REGION Network 21: PM1 Count & CycleTime / PM19 Count & CycleTime
   RUNG wire#powerrail
      #PM19CountCycleTime(iAlwaysOn := #iAlwaysOn, iProcessStart := "ST10_PM".Num[19].ProcessStart, iProcessComplete := "ST10_PM".Num[19].ProcessComplete, iProcessResult := "ST10_PM".Num[19].ProcessResult, ioCount := "ST10_PMCountCycleTime".PM[19].Count, ioTotalCycleTime := "ST10_PMCountCycleTime".PM[19].TotalCycleTime, ioMachineCycleTime := "ST10_PMCountCycleTime".PM[19].MachineCycleTime)
   END_RUNG
   // the same network as SCL:
   #PM19CountCycleTime(iAlwaysOn := #iAlwaysOn,   // "Count_CycleTime_V3"
                       iProcessStart := "ST10_PM".Num[19].ProcessStart,
                       iProcessComplete := "ST10_PM".Num[19].ProcessComplete,
                       iProcessResult := "ST10_PM".Num[19].ProcessResult,
                       ioCount := "ST10_PMCountCycleTime".PM[19].Count,
                       ioTotalCycleTime := "ST10_PMCountCycleTime".PM[19].TotalCycleTime,
                       ioMachineCycleTime := "ST10_PMCountCycleTime".PM[19].MachineCycleTime);
END_REGION

REGION Network 22: PM2 Count & CycleTime / PM20 Count & CycleTime
   RUNG wire#powerrail
      #PM20CountCycleTime(iAlwaysOn := #iAlwaysOn, iProcessStart := "ST10_PM".Num[20].ProcessStart, iProcessComplete := "ST10_PM".Num[20].ProcessComplete, iProcessResult := "ST10_PM".Num[20].ProcessResult, ioCount := "ST10_PMCountCycleTime".PM[20].Count, ioTotalCycleTime := "ST10_PMCountCycleTime".PM[20].TotalCycleTime, ioMachineCycleTime := "ST10_PMCountCycleTime".PM[20].MachineCycleTime)
   END_RUNG
   // the same network as SCL:
   #PM20CountCycleTime(iAlwaysOn := #iAlwaysOn,   // "Count_CycleTime_V3"
                       iProcessStart := "ST10_PM".Num[20].ProcessStart,
                       iProcessComplete := "ST10_PM".Num[20].ProcessComplete,
                       iProcessResult := "ST10_PM".Num[20].ProcessResult,
                       ioCount := "ST10_PMCountCycleTime".PM[20].Count,
                       ioTotalCycleTime := "ST10_PMCountCycleTime".PM[20].TotalCycleTime,
                       ioMachineCycleTime := "ST10_PMCountCycleTime".PM[20].MachineCycleTime);
END_REGION

REGION Network 23: PM2 Count & CycleTime / PM21 Count & CycleTime
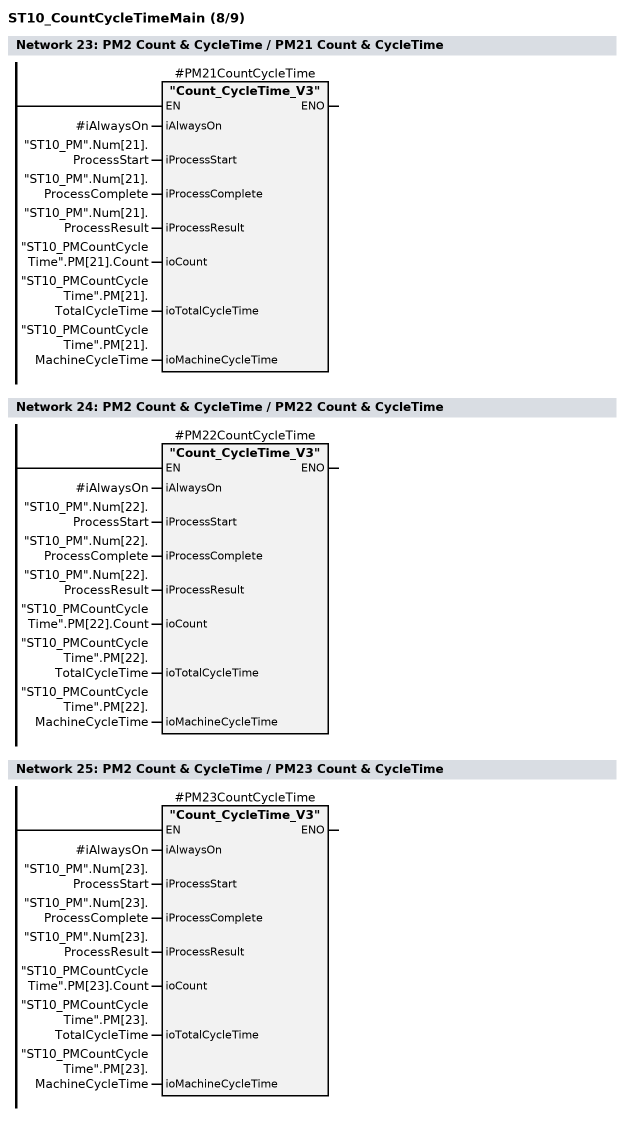
   RUNG wire#powerrail
      #PM21CountCycleTime(iAlwaysOn := #iAlwaysOn, iProcessStart := "ST10_PM".Num[21].ProcessStart, iProcessComplete := "ST10_PM".Num[21].ProcessComplete, iProcessResult := "ST10_PM".Num[21].ProcessResult, ioCount := "ST10_PMCountCycleTime".PM[21].Count, ioTotalCycleTime := "ST10_PMCountCycleTime".PM[21].TotalCycleTime, ioMachineCycleTime := "ST10_PMCountCycleTime".PM[21].MachineCycleTime)
   END_RUNG
   // the same network as SCL:
   #PM21CountCycleTime(iAlwaysOn := #iAlwaysOn,   // "Count_CycleTime_V3"
                       iProcessStart := "ST10_PM".Num[21].ProcessStart,
                       iProcessComplete := "ST10_PM".Num[21].ProcessComplete,
                       iProcessResult := "ST10_PM".Num[21].ProcessResult,
                       ioCount := "ST10_PMCountCycleTime".PM[21].Count,
                       ioTotalCycleTime := "ST10_PMCountCycleTime".PM[21].TotalCycleTime,
                       ioMachineCycleTime := "ST10_PMCountCycleTime".PM[21].MachineCycleTime);
END_REGION

REGION Network 24: PM2 Count & CycleTime / PM22 Count & CycleTime
   RUNG wire#powerrail
      #PM22CountCycleTime(iAlwaysOn := #iAlwaysOn, iProcessStart := "ST10_PM".Num[22].ProcessStart, iProcessComplete := "ST10_PM".Num[22].ProcessComplete, iProcessResult := "ST10_PM".Num[22].ProcessResult, ioCount := "ST10_PMCountCycleTime".PM[22].Count, ioTotalCycleTime := "ST10_PMCountCycleTime".PM[22].TotalCycleTime, ioMachineCycleTime := "ST10_PMCountCycleTime".PM[22].MachineCycleTime)
   END_RUNG
   // the same network as SCL:
   #PM22CountCycleTime(iAlwaysOn := #iAlwaysOn,   // "Count_CycleTime_V3"
                       iProcessStart := "ST10_PM".Num[22].ProcessStart,
                       iProcessComplete := "ST10_PM".Num[22].ProcessComplete,
                       iProcessResult := "ST10_PM".Num[22].ProcessResult,
                       ioCount := "ST10_PMCountCycleTime".PM[22].Count,
                       ioTotalCycleTime := "ST10_PMCountCycleTime".PM[22].TotalCycleTime,
                       ioMachineCycleTime := "ST10_PMCountCycleTime".PM[22].MachineCycleTime);
END_REGION

REGION Network 25: PM2 Count & CycleTime / PM23 Count & CycleTime
   RUNG wire#powerrail
      #PM23CountCycleTime(iAlwaysOn := #iAlwaysOn, iProcessStart := "ST10_PM".Num[23].ProcessStart, iProcessComplete := "ST10_PM".Num[23].ProcessComplete, iProcessResult := "ST10_PM".Num[23].ProcessResult, ioCount := "ST10_PMCountCycleTime".PM[23].Count, ioTotalCycleTime := "ST10_PMCountCycleTime".PM[23].TotalCycleTime, ioMachineCycleTime := "ST10_PMCountCycleTime".PM[23].MachineCycleTime)
   END_RUNG
   // the same network as SCL:
   #PM23CountCycleTime(iAlwaysOn := #iAlwaysOn,   // "Count_CycleTime_V3"
                       iProcessStart := "ST10_PM".Num[23].ProcessStart,
                       iProcessComplete := "ST10_PM".Num[23].ProcessComplete,
                       iProcessResult := "ST10_PM".Num[23].ProcessResult,
                       ioCount := "ST10_PMCountCycleTime".PM[23].Count,
                       ioTotalCycleTime := "ST10_PMCountCycleTime".PM[23].TotalCycleTime,
                       ioMachineCycleTime := "ST10_PMCountCycleTime".PM[23].MachineCycleTime);
END_REGION

REGION Network 26: PM2 Count & CycleTime / PM24 Count & CycleTime
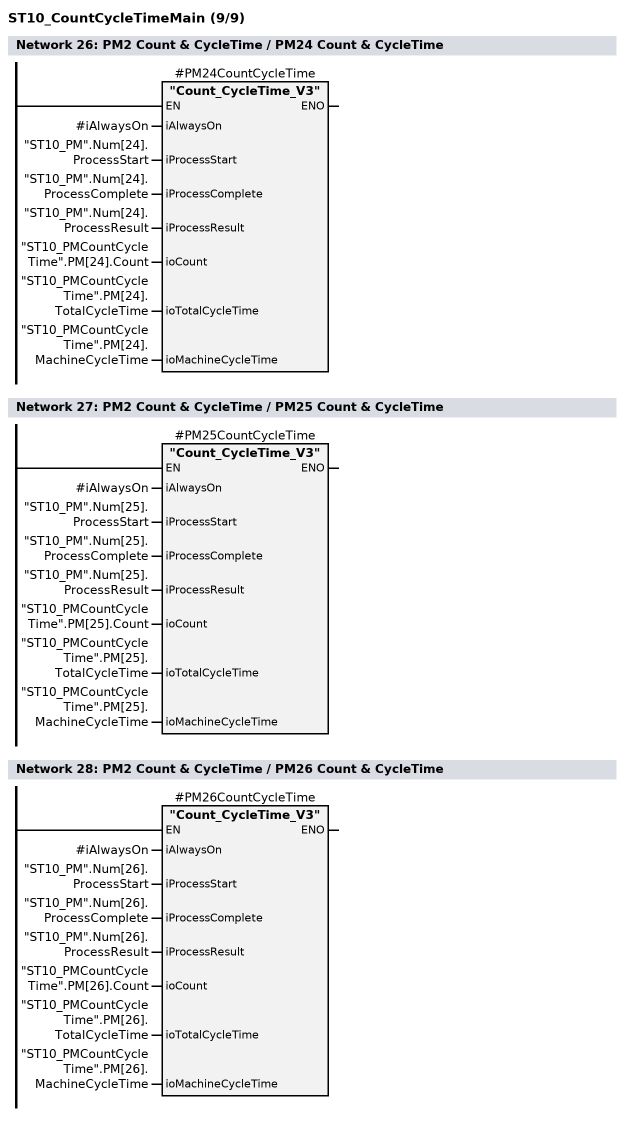
   RUNG wire#powerrail
      #PM24CountCycleTime(iAlwaysOn := #iAlwaysOn, iProcessStart := "ST10_PM".Num[24].ProcessStart, iProcessComplete := "ST10_PM".Num[24].ProcessComplete, iProcessResult := "ST10_PM".Num[24].ProcessResult, ioCount := "ST10_PMCountCycleTime".PM[24].Count, ioTotalCycleTime := "ST10_PMCountCycleTime".PM[24].TotalCycleTime, ioMachineCycleTime := "ST10_PMCountCycleTime".PM[24].MachineCycleTime)
   END_RUNG
   // the same network as SCL:
   #PM24CountCycleTime(iAlwaysOn := #iAlwaysOn,   // "Count_CycleTime_V3"
                       iProcessStart := "ST10_PM".Num[24].ProcessStart,
                       iProcessComplete := "ST10_PM".Num[24].ProcessComplete,
                       iProcessResult := "ST10_PM".Num[24].ProcessResult,
                       ioCount := "ST10_PMCountCycleTime".PM[24].Count,
                       ioTotalCycleTime := "ST10_PMCountCycleTime".PM[24].TotalCycleTime,
                       ioMachineCycleTime := "ST10_PMCountCycleTime".PM[24].MachineCycleTime);
END_REGION

REGION Network 27: PM2 Count & CycleTime / PM25 Count & CycleTime
   RUNG wire#powerrail
      #PM25CountCycleTime(iAlwaysOn := #iAlwaysOn, iProcessStart := "ST10_PM".Num[25].ProcessStart, iProcessComplete := "ST10_PM".Num[25].ProcessComplete, iProcessResult := "ST10_PM".Num[25].ProcessResult, ioCount := "ST10_PMCountCycleTime".PM[25].Count, ioTotalCycleTime := "ST10_PMCountCycleTime".PM[25].TotalCycleTime, ioMachineCycleTime := "ST10_PMCountCycleTime".PM[25].MachineCycleTime)
   END_RUNG
   // the same network as SCL:
   #PM25CountCycleTime(iAlwaysOn := #iAlwaysOn,   // "Count_CycleTime_V3"
                       iProcessStart := "ST10_PM".Num[25].ProcessStart,
                       iProcessComplete := "ST10_PM".Num[25].ProcessComplete,
                       iProcessResult := "ST10_PM".Num[25].ProcessResult,
                       ioCount := "ST10_PMCountCycleTime".PM[25].Count,
                       ioTotalCycleTime := "ST10_PMCountCycleTime".PM[25].TotalCycleTime,
                       ioMachineCycleTime := "ST10_PMCountCycleTime".PM[25].MachineCycleTime);
END_REGION

REGION Network 28: PM2 Count & CycleTime / PM26 Count & CycleTime
   RUNG wire#powerrail
      #PM26CountCycleTime(iAlwaysOn := #iAlwaysOn, iProcessStart := "ST10_PM".Num[26].ProcessStart, iProcessComplete := "ST10_PM".Num[26].ProcessComplete, iProcessResult := "ST10_PM".Num[26].ProcessResult, ioCount := "ST10_PMCountCycleTime".PM[26].Count, ioTotalCycleTime := "ST10_PMCountCycleTime".PM[26].TotalCycleTime, ioMachineCycleTime := "ST10_PMCountCycleTime".PM[26].MachineCycleTime)
   END_RUNG
   // the same network as SCL:
   #PM26CountCycleTime(iAlwaysOn := #iAlwaysOn,   // "Count_CycleTime_V3"
                       iProcessStart := "ST10_PM".Num[26].ProcessStart,
                       iProcessComplete := "ST10_PM".Num[26].ProcessComplete,
                       iProcessResult := "ST10_PM".Num[26].ProcessResult,
                       ioCount := "ST10_PMCountCycleTime".PM[26].Count,
                       ioTotalCycleTime := "ST10_PMCountCycleTime".PM[26].TotalCycleTime,
                       ioMachineCycleTime := "ST10_PMCountCycleTime".PM[26].MachineCycleTime);
END_REGION
END_FUNCTION_BLOCK

FUNCTION_BLOCK "Count_CycleTime"   // FB3002, SCL
TITLE = Count_CycleTime
{ S7_Optimized_Access := 'TRUE' }
AUTHOR : STD
FAMILY : RCS
VERSION : 18.0
// 1.count
// 2.cycle time
// stored: AutoNumber false, MemoryReserve 100, SetENOAutomatically false, UDAEnableTagReadback true
   VAR_INPUT
      iAlwaysOn : Bool;
      iRun : Bool;
      iManualMode : Bool;
      iAutoMode : Bool;
      iAutoRunning : Bool;
      iProcessStart : Bool;
      iProcessComplete : Bool;
      iProcessResult : DInt;
   END_VAR
   VAR_IN_OUT
      ioCount : "RCS_SysCount_V1";
      ioTotalCycleTime : "RCS_SysCycleTime_V1";
      ioMachineCycleTime : "RCS_SysCycleTime_V1";
   END_VAR
   VAR
      sFlow : Struct
         pls : Array[0..15] of Bool;
         sDTStart : Date_And_Time;
         sDTRes : Date_And_Time;
         sDTOld : Date_And_Time;
         sDTRuntime : Date_And_Time;
         sDTRunning : Date_And_Time;
         sDTCurrent : Date_And_Time;
         Run_Minute : Int;
         Run_Hour : Int;
         Run_Day : Int;
         AutoRun_Minute : Int;
         AutoRun_Hour : Int;
         AutoRun_Day : Int;
      END_STRUCT;
   END_VAR
   VAR_TEMP
      tStart : Bool;
      tStop : Bool;
      tAutorunning : Bool;
      tpt : Int;
      tpRet : Int;
      tpResult : Time;
      tDint : DInt;
      tReal : Array[0..1] of Real;
   END_VAR
BEGIN
   (*############################################################
      RUHLAMAT SUZHOU ELEC.STD.
      Copyright (c) 2017. All rights reserved.    

      NAME OF FUNCTION BLOCK:         Count_CycleTimeV2.0
      VERSION NUMBER:                 V2.0
      COMPOSER:                       Ming.Jiang

      LAST CHANGE:                    13.April.2017
      Comment by Ming.Jiang 

      #RET_VALUE:


      #Alert Value:



      -----------------------------------------------------
      Date        Name      Version           Activity                                                                              

   ############################################################*)

   #tStart := #iProcessStart AND NOT #sFlow.pls[0];
   #sFlow.pls[0] := #iProcessStart;
   #tStop := #iProcessComplete AND NOT #sFlow.pls[1];
   #sFlow.pls[1] := #iProcessComplete;
   #tAutorunning := #iAutoMode AND #iAutoRunning AND NOT #sFlow.pls[2];
   #sFlow.pls[2] := #iAutoRunning AND #iAutoMode;

   IF #tAutorunning THEN
       #tpRet := RD_SYS_T(#sFlow.sDTOld);
   END_IF;

   //Machine Cycle time
   IF #iAutoMode AND NOT #iManualMode AND #iAutoRunning THEN
       IF #tStart THEN
           #tpRet := RD_SYS_T(#sFlow.sDTStart);
       END_IF;
       IF #tStop THEN

           //MachineTime
           #ioMachineCycleTime.No[21] := 0.0;
           #tpRet := RD_SYS_T(#sFlow.sDTRes);
           #tReal[0] := DINT_TO_REAL(TIME_TO_DINT(T_DIFF(IN1 := #sFlow.sDTRes, IN2 :=#sFlow.sDTStart )));
           #ioMachineCycleTime.No[0] :=  #tReal[0]/1000.0;

           //TotalTime
           #ioTotalCycleTime.No[21] := 0.0;
           #tReal[1] := DINT_TO_REAL(TIME_TO_DINT(T_DIFF(IN1 := #sFlow.sDTRes, IN2 := #sFlow.sDTOld)));
           #tpRet := RD_SYS_T(#sFlow.sDTOld);
           #ioTotalCycleTime.No[0] := #tReal[1]/1000.0;
           FOR #tpt := 20 TO 1 BY -1  DO
               //MachineTime
               #ioMachineCycleTime.No[#tpt] := #ioMachineCycleTime.No[#tpt - 1];
               #ioMachineCycleTime.No[21] := #ioMachineCycleTime.No[21] + #ioMachineCycleTime.No[#tpt];
               //totalCycleTime
               #ioTotalCycleTime.No[#tpt] := #ioTotalCycleTime.No[#tpt - 1];
               #ioTotalCycleTime.No[21] := #ioTotalCycleTime.No[21] + #ioTotalCycleTime.No[#tpt];
           END_FOR;
           //MachineTime
           #ioMachineCycleTime.No[21] := #ioMachineCycleTime.No[21] / 20.0;
           //totalCycleTime
           #ioTotalCycleTime.No[21] := #ioTotalCycleTime.No[21] / 20.0;

           //Count-------------------------------------------------------//
           IF #iProcessResult = 400 THEN
               #ioCount.OK[0] := #ioCount.OK[0] + 1;
               #ioCount.OKHolding := #ioCount.OKHolding + 1;
           END_IF;
           IF #iProcessResult > 400  THEN
               #ioCount.NG[0] := #ioCount.NG[0] + 1;
               #ioCount.NGHolding:=#ioCount.NGHolding+1;
           END_IF;
           IF #iProcessResult >=400  THEN
               #ioCount.Total := #ioCount.Total + 1;
           END_IF;
           #ioCount.OKHolding := #ioCount.OKHolding + 1;

           CASE #iProcessResult OF
               401:  //NG1
                   #ioCount.NG[1] := #ioCount.NG[1] + 1;
               402:  //NG1uuuuuuuuuuuuuuuuuuuuuuuuuuuuuuuuuuuuuuuuuuuuuuuu
                   #ioCount.NG[2] := #ioCount.NG[2] + 1;
               403:  //NG1uuuuu
                   #ioCount.NG[3] := #ioCount.NG[3] + 1;
               404:  //NG1
                   #ioCount.NG[4] := #ioCount.NG[4] + 1;
               405:  //NG1
                   #ioCount.NG[5] := #ioCount.NG[5] + 1;
               406:  //NG1
                   #ioCount.NG[6] := #ioCount.NG[6] + 1;
               407:  //NG1
                   #ioCount.NG[7] := #ioCount.NG[7] + 1;
               408:  //NG1
                   #ioCount.NG[8] := #ioCount.NG[8] + 1;
               409:  //NG1
                   #ioCount.NG[9] := #ioCount.NG[9] + 1;

           END_CASE;
       END_IF;

   END_IF;
   //clear 
   IF #ioCount.ClearOK AND NOT #sFlow.pls[3] THEN
       #ioCount.OK[0] := 0;

   END_IF;
   #sFlow.pls[3] := #ioCount.ClearOK;
   IF #ioCount.ClearNG AND NOT #sFlow.pls[4] THEN
       FOR #tpt := 0 TO 9 DO
            #ioCount.NG[#tpt] := 0;
        END_FOR;
   END_IF;
   #sFlow.pls[4] := #ioCount.ClearNG;
   IF #ioCount.ClearTotal AND NOT #sFlow.pls[5] THEN
       #ioCount.Total := 0;

   END_IF;
   #sFlow.pls[5] := #ioCount.ClearTotal;
   //Runtime

   IF #iAutoRunning AND NOT #sFlow.pls[6] THEN
       #tpRet := RD_SYS_T(#sFlow.sDTRunning);

   END_IF;
   #sFlow.pls[6] := #iAutoRunning;
   #tpRet := RD_SYS_T(#sFlow.sDTCurrent);
   IF #iAutoRunning THEN
       #tDint := TIME_TO_DINT(T_DIFF(IN1 := #sFlow.sDTCurrent, IN2 := #sFlow.sDTRunning));
       #tReal[0] := DINT_TO_REAL(#tDint) / 1000.0;
       #sFlow.AutoRun_Day := REAL_TO_INT(#tReal[0] / 86400.0);
       #sFlow.AutoRun_Hour := (REAL_TO_DINT(#tReal[0]) MOD 86400) / 3600;
       #sFlow.AutoRun_Minute := ((REAL_TO_DINT(#tReal[0]) MOD 86400) MOD 3600) / 60;
   END_IF;

   //Runtime
   IF #iRun AND NOT #sFlow.pls[7] THEN
       #tpRet := RD_SYS_T(#sFlow.sDTRuntime);
   END_IF;
   #sFlow.pls[7] := #iRun;
   IF #iRun THEN
       #tDint := TIME_TO_DINT(T_DIFF(IN1 := #sFlow.sDTCurrent, IN2 :=#sFlow.sDTRuntime ));
       #tReal[0] := DINT_TO_REAL(#tDint) / 1000.0;
       #sFlow.Run_Day := REAL_TO_INT(#tReal[0] / 86400.0);
       #sFlow.Run_Hour := (REAL_TO_DINT(#tReal[0]) MOD 86400) / 3600;
       #sFlow.Run_Minute := ((REAL_TO_DINT(#tReal[0]) MOD 86400) MOD 3600) / 60;
   END_IF;
END_FUNCTION_BLOCK

FUNCTION_BLOCK "Count_CycleTime_V3"   // FB3003, SCL
TITLE = Count_CycleTime
{ S7_Optimized_Access := 'TRUE' }
AUTHOR : STD
FAMILY : RCS
VERSION : 18.0
// 1.count
// 2.cycle time
// stored: AutoNumber false, MemoryReserve 100, SetENOAutomatically false, UDAEnableTagReadback true
   VAR_INPUT
      iAlwaysOn : Bool;
      iProcessStart : Bool;
      iProcessComplete : Bool;
      iProcessResult : DInt;
   END_VAR
   VAR_IN_OUT
      ioCount : "RCS_SysCount_V1";
      ioTotalCycleTime : "RCS_SysCycleTime_V1";
      ioMachineCycleTime : "RCS_SysCycleTime_V1";
   END_VAR
   VAR
      sFlow : Struct
         pls : Array[0..15] of Bool;
         sDTStart : Date_And_Time;
         sDTRes : Date_And_Time;
         sDTOld : Date_And_Time;
         sDTRuntime : Date_And_Time;
         sDTRunning : Date_And_Time;
         sDTCurrent : Date_And_Time;
         Run_Minute : Int;
         Run_Hour : Int;
         Run_Day : Int;
         AutoRun_Minute : Int;
         AutoRun_Hour : Int;
         AutoRun_Day : Int;
      END_STRUCT;
   END_VAR
   VAR_TEMP
      tStart : Bool;
      tStop : Bool;
      tAutorunning : Bool;
      tpt : Int;
      tpRet : Int;
      tpResult : Time;
      tDint : DInt;
      tReal : Array[0..1] of Real;
   END_VAR
BEGIN
   (*############################################################
      RUHLAMAT SUZHOU ELEC.STD.
      Copyright (c) 2017. All rights reserved.    

      NAME OF FUNCTION BLOCK:         Count_CycleTimeV2.0
      VERSION NUMBER:                 V2.0
      COMPOSER:                       Ming.Jiang

      LAST CHANGE:                    13.April.2017
      Comment by Ming.Jiang 

      #RET_VALUE:


      #Alert Value:



      -----------------------------------------------------
      Date        Name      Version           Activity                                                                              

   ############################################################*)

   #tStart := #iProcessStart AND NOT #sFlow.pls[0];
   #sFlow.pls[0] := #iProcessStart;
   #tStop := #iProcessComplete AND NOT #sFlow.pls[1];
   #sFlow.pls[1] := #iProcessComplete;

   // IF #tStop THEN
   //     #tpRet := RD_SYS_T(#sFlow.sDTOld);
   // END_IF;

   //Machine Cycle time
   IF TRUE THEN
       IF #tStart THEN
           #tpRet := RD_SYS_T(#sFlow.sDTStart);
       END_IF;
       IF #tStop THEN

           //MachineTime
           #ioMachineCycleTime.No[21] := 0.0;
           #tpRet := RD_SYS_T(#sFlow.sDTRes);
           #tReal[0] := DINT_TO_REAL(TIME_TO_DINT(T_DIFF(IN1 := #sFlow.sDTRes, IN2 :=#sFlow.sDTStart )));
           #ioMachineCycleTime.No[0] :=  #tReal[0]/1000.0;

           //TotalTime
           #ioTotalCycleTime.No[21] := 0.0;
           #tReal[1] := DINT_TO_REAL(TIME_TO_DINT(T_DIFF(IN1 := #sFlow.sDTRes, IN2 := #sFlow.sDTOld)));
           #tpRet := RD_SYS_T(#sFlow.sDTOld);
           #ioTotalCycleTime.No[0] := #tReal[1]/1000.0;
           FOR #tpt := 20 TO 1 BY -1  DO
               //MachineTime
               #ioMachineCycleTime.No[#tpt] := #ioMachineCycleTime.No[#tpt - 1];
               #ioMachineCycleTime.No[21] := #ioMachineCycleTime.No[21] + #ioMachineCycleTime.No[#tpt];
               //totalCycleTime
               #ioTotalCycleTime.No[#tpt] := #ioTotalCycleTime.No[#tpt - 1];
               #ioTotalCycleTime.No[21] := #ioTotalCycleTime.No[21] + #ioTotalCycleTime.No[#tpt];
           END_FOR;
           //MachineTime
           #ioMachineCycleTime.No[21] := #ioMachineCycleTime.No[21] / 20.0;
           //totalCycleTime
           #ioTotalCycleTime.No[21] := #ioTotalCycleTime.No[21] / 20.0;

           //Count-------------------------------------------------------//
           IF #iProcessResult = 400 THEN
               #ioCount.OK[0] := #ioCount.OK[0] + 1;
               #ioCount.OKHolding := #ioCount.OKHolding + 1;
           END_IF;
           IF #iProcessResult >400 THEN
               #ioCount.NG[0] := #ioCount.NG[0] + 1;
               #ioCount.NGHolding:=#ioCount.NGHolding+1;
           END_IF;
           IF #iProcessResult >=400 THEN
               #ioCount.Total := #ioCount.Total + 1;
           END_IF;
           #ioCount.OKHolding := #ioCount.OKHolding + 1;

           CASE #iProcessResult OF
               401:  //NG1
                   #ioCount.NG[1] := #ioCount.NG[1] + 1;
               402:  //NG1uuuuuuuuuuuuuuuuuuuuuuuuuuuuuuuuuuuuuuuuuuuuuuuu
                   #ioCount.NG[2] := #ioCount.NG[2] + 1;
               403:  //NG1uuuuu
                   #ioCount.NG[3] := #ioCount.NG[3] + 1;
               404:  //NG1
                   #ioCount.NG[4] := #ioCount.NG[4] + 1;
               405:  //NG1
                   #ioCount.NG[5] := #ioCount.NG[5] + 1;
               406:  //NG1
                   #ioCount.NG[6] := #ioCount.NG[6] + 1;
               407:  //NG1
                   #ioCount.NG[7] := #ioCount.NG[7] + 1;
               408:  //NG1
                   #ioCount.NG[8] := #ioCount.NG[8] + 1;
               409:  //NG1
                   #ioCount.NG[9] := #ioCount.NG[9] + 1;

           END_CASE;
       END_IF;

   END_IF;
   //clear 
   IF #ioCount.ClearOK AND NOT #sFlow.pls[3] THEN
       #ioCount.OK[0] := 0;

   END_IF;
   #sFlow.pls[3] := #ioCount.ClearOK;
   IF #ioCount.ClearNG AND NOT #sFlow.pls[4] THEN
       FOR #tpt := 0 TO 9 DO
            #ioCount.NG[#tpt] := 0;
        END_FOR;
   END_IF;
   #sFlow.pls[4] := #ioCount.ClearNG;
   IF #ioCount.ClearTotal AND NOT #sFlow.pls[5] THEN
       #ioCount.Total := 0;

   END_IF;
   #sFlow.pls[5] := #ioCount.ClearTotal;
END_FUNCTION_BLOCK

FUNCTION_BLOCK "SystemMode"   // FB3000, LAD
TITLE = SystemMode_FB
{ S7_Optimized_Access := 'TRUE' }
AUTHOR : STD
FAMILY : RCS
VERSION : 2.0
// stored: AutoNumber false, MemoryReserve 100, SetENOAutomatically false
   VAR_INPUT
      iPLCRestarted : Bool;
      iEstopAllOK { ExternalAccessible := 'False'; ExternalVisible := 'False'; ExternalWritable := 'False'} : Bool;   // 急停按钮
      iResetFault { ExternalAccessible := 'False'; ExternalVisible := 'False'; ExternalWritable := 'False'} : Bool;   // 故障复位按钮
      iModeSelectType { ExternalAccessible := 'False'; ExternalVisible := 'False'; ExternalWritable := 'False'} : Bool;   // 0=key switch / 1= HMI button
      iManual { ExternalAccessible := 'False'; ExternalVisible := 'False'; ExternalWritable := 'False'} : Bool;   // Key switch signal,1=Manual / Key switch signal,1=Manual Mode
      iAuto { ExternalAccessible := 'False'; ExternalVisible := 'False'; ExternalWritable := 'False'} : Bool;   // Key switch signal,1=Auto / Key switch signal,1=Auto Mode
      iStep { ExternalAccessible := 'False'; ExternalVisible := 'False'; ExternalWritable := 'False'} : Bool;   // Step mode / Auto Step Mode
      iOneCycle : Bool;   // OneCycle / Auto One Cycle Mode
      iHMIModeSelect { ExternalAccessible := 'False'; ExternalVisible := 'False'; ExternalWritable := 'False'} : Int;   // HMI button signal,1=Manual / 2=Auto/3=OneCycle/4=Step / HMI button signal,1=Manual / 2=Auto / 3=Step / 4=OneCyc
      iControlOnMonitor { ExternalAccessible := 'False'; ExternalVisible := 'False'; ExternalWritable := 'False'} : Bool;   // 安全继电器ControlOn监控
      iSafetyDoor { ExternalAccessible := 'False'; ExternalVisible := 'False'; ExternalWritable := 'False'} : Bool;
      iLightCurtain { ExternalAccessible := 'False'; ExternalVisible := 'False'; ExternalWritable := 'False'} : Bool;
      iSafetyByPass : Bool;
      iMainPressureSwitch { ExternalAccessible := 'False'; ExternalVisible := 'False'; ExternalWritable := 'False'} : Bool;   // 主气源开关监控
      iFixtureOK { ExternalAccessible := 'False'; ExternalVisible := 'False'; ExternalWritable := 'False'} : Bool;   // fixture ok
      iChangeOverOK { ExternalAccessible := 'False'; ExternalVisible := 'False'; ExternalWritable := 'False'} : Bool;   // changer over is ok
      iInitializationOK { ExternalAccessible := 'False'; ExternalVisible := 'False'; ExternalWritable := 'False'} : Bool;   // initialization is ok
      iAllDeviceOK { ExternalAccessible := 'False'; ExternalVisible := 'False'; ExternalWritable := 'False'} : Bool;   // all device is ready
      iAlarmOn : Bool;   // 设备故障
      iFlowRun : Bool;   // 设备运行
   END_VAR
   VAR_OUTPUT
      oReset { ExternalAccessible := 'False'; ExternalVisible := 'False'; ExternalWritable := 'False'} : Bool;   // 系统复位信号
      oEStopOK { ExternalAccessible := 'False'; ExternalVisible := 'False'; ExternalWritable := 'False'} : Bool;   // 系统急停控制信号
      oManualMode { ExternalAccessible := 'False'; ExternalVisible := 'False'; ExternalWritable := 'False'} : Bool;   // 手动模式信号
      oAutoMode { ExternalAccessible := 'False'; ExternalVisible := 'False'; ExternalWritable := 'False'} : Bool;   // 自动模式信号
      oOneCycleMode : Bool;   // 单次循环
      oStepMode { ExternalAccessible := 'False'; ExternalVisible := 'False'; ExternalWritable := 'False'} : Bool;
      oRun { ExternalAccessible := 'False'; ExternalVisible := 'False'; ExternalWritable := 'False'} : Bool;   // 系统运行就绪信号 / Control On and all Safety function OK
      "oEnable alarm" : Bool;
      oControlON { ExternalAccessible := 'False'; ExternalVisible := 'False'; ExternalWritable := 'False'} : Bool;   // PowerON
      oMainPressureOK { ExternalAccessible := 'False'; ExternalVisible := 'False'; ExternalWritable := 'False'} : Bool;   // air pressure
      oSafetyDoorOK { ExternalAccessible := 'False'; ExternalVisible := 'False'; ExternalWritable := 'False'} : Bool;   // 安全门关闭
      oLightCurtainOK { ExternalAccessible := 'False'; ExternalVisible := 'False'; ExternalWritable := 'False'} : Bool;   // 光栅
      oReady : Bool;   // 用于流程控制 / In AutoMode and all condition ok, machine can auto running
      oMode { ExternalAccessible := 'False'; ExternalVisible := 'False'; ExternalWritable := 'False'} : Int;   // 0NA,1Manual, 2Auto, 3Step, 4OneCycle, 5Runn, 6Error
      oStatus : Int;   // 0NotReady, 1Ready, 2AutoRunning, 3EStop, 4Alarm
   END_VAR
   VAR
      sRunT { S7_SetPoint := 'True'} : TON_TIME;
      sPressureTOF { S7_SetPoint := 'True'} : TOF_TIME;
      sChangeOverTOF { S7_SetPoint := 'True'} : TOF_TIME;
      sChangeOverOK { S7_SetPoint := 'True'} : Bool;
   END_VAR
   VAR_TEMP
      tAlwaysOn : Bool;
   END_VAR
   VAR_TEMP   // added for the SCL form of the ladder/FBD networks
      _w1 : Bool;
      _w2 : Bool;
      _w3 : Bool;
   END_VAR
BEGIN

REGION Network 1: AlwaysOn
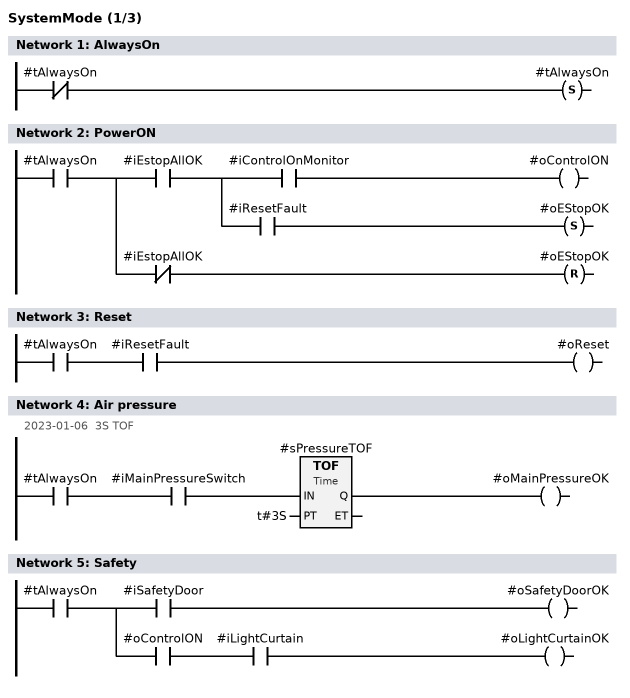
   RUNG wire#powerrail
      I_Contact( #tAlwaysOn )
      S_Coil( #tAlwaysOn )
   END_RUNG
   // the same network as SCL:
   IF NOT #tAlwaysOn THEN #tAlwaysOn := TRUE; END_IF;
END_REGION

REGION Network 2: PowerON
   RUNG wire#powerrail
      Contact( #tAlwaysOn )
      wire#w1
      Contact( #iEstopAllOK )
      wire#w2
      Contact( #iControlOnMonitor )
      Coil( #oControlON )
   END_RUNG
   RUNG wire#w2
      Contact( #iResetFault )
      S_Coil( #oEStopOK )
   END_RUNG
   RUNG wire#w1
      I_Contact( #iEstopAllOK )
      R_Coil( #oEStopOK )
   END_RUNG
   // the same network as SCL:
   #_w1 := #tAlwaysOn AND #iEstopAllOK;
   #oControlON := #_w1 AND #iControlOnMonitor;
   IF #_w1 AND #iResetFault THEN #oEStopOK := TRUE; END_IF;
   IF #tAlwaysOn AND NOT #iEstopAllOK THEN #oEStopOK := FALSE; END_IF;
END_REGION

REGION Network 3: Reset
   RUNG wire#powerrail
      Contact( #tAlwaysOn )
      Contact( #iResetFault )
      Coil( #oReset )
   END_RUNG
   // the same network as SCL:
   #oReset := #tAlwaysOn AND #iResetFault;
END_REGION

REGION Network 4: Air pressure
   // 2023-01-06  3S TOF
   RUNG wire#powerrail
      Contact( #tAlwaysOn )
      Contact( #iMainPressureSwitch )
      { S7_Templates := "time_type := Time" } #sPressureTOF.TOF(pt := t#3S, et =>)
      Coil( #oMainPressureOK )
   END_RUNG
   // the same network as SCL:
   #sPressureTOF(IN := #tAlwaysOn AND #iMainPressureSwitch, PT := t#3S);   // TOF
   #oMainPressureOK := #sPressureTOF.Q;
END_REGION

REGION Network 5: Safety
   RUNG wire#powerrail
      Contact( #tAlwaysOn )
      wire#w1
      Contact( #iSafetyDoor )
      Coil( #oSafetyDoorOK )
   END_RUNG
   RUNG wire#w1
      Contact( #oControlON )
      Contact( #iLightCurtain )
      Coil( #oLightCurtainOK )
   END_RUNG
   // the same network as SCL:
   #oSafetyDoorOK := #tAlwaysOn AND #iSafetyDoor;
   #oLightCurtainOK := #tAlwaysOn AND #oControlON AND #iLightCurtain;
END_REGION

REGION Network 6: Mode
   // 0NA,1Manual, 2Auto, 3Step, 4OneCycle, 5Runn, 6Error
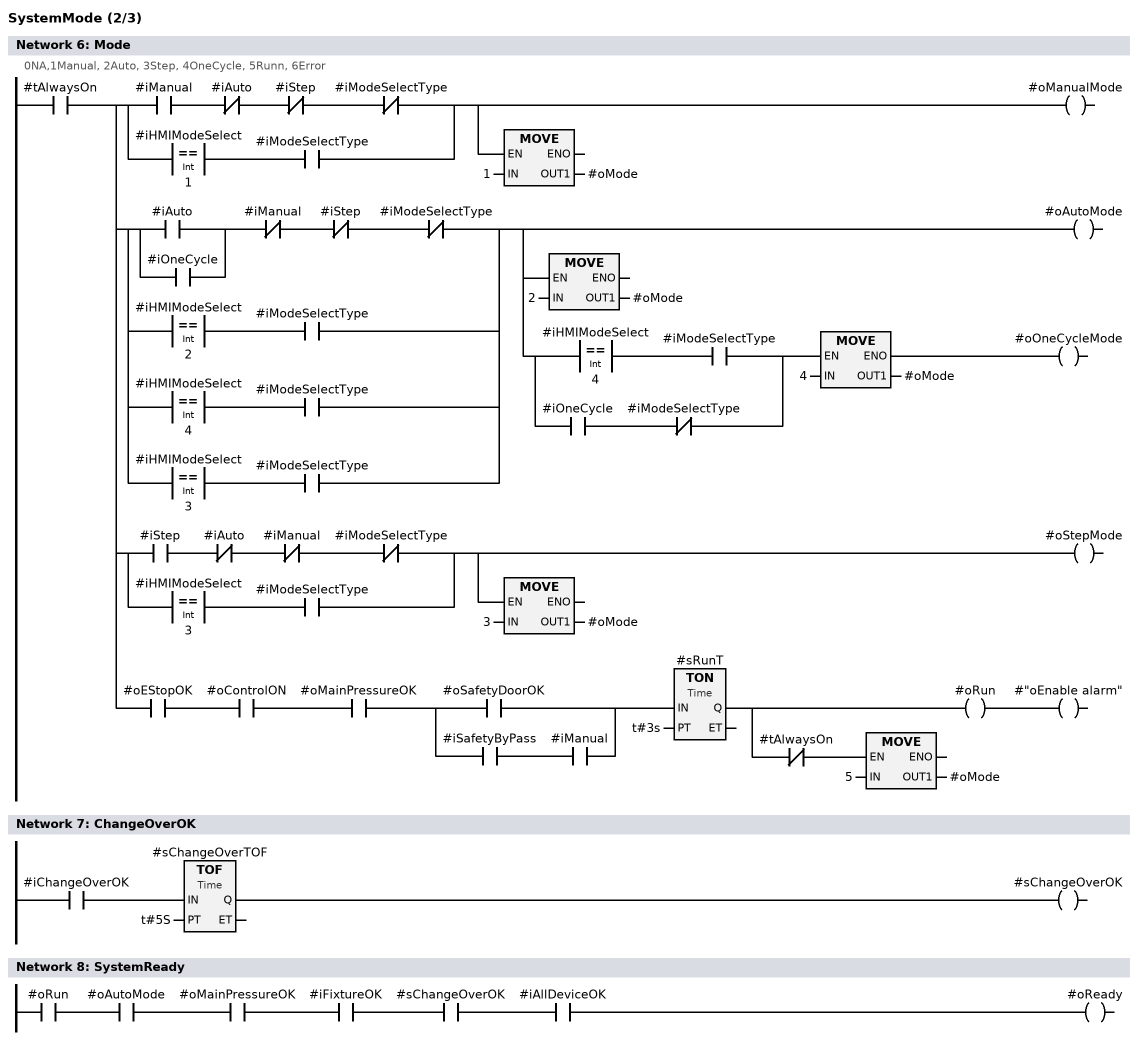
   RUNG wire#powerrail
      Contact( #tAlwaysOn )
      wire#w1
      Contact( #iManual )
      I_Contact( #iAuto )
      I_Contact( #iStep )
      I_Contact( #iModeSelectType )
      wire#w2
      Coil( #oManualMode )
   END_RUNG
   RUNG wire#w1
      { S7_Templates := "SrcType := Int" } EQ_Contact(in1 := #iHMIModeSelect, in2 := 1)
      Contact( #iModeSelectType )
   END_RUNG wire#w2
   RUNG wire#w2
      { S7_GenerateENO := "TRUE" } Move(in := 1, out1 => #oMode)
   END_RUNG
   RUNG wire#w1
      Contact( #iAuto )
      wire#w3
      I_Contact( #iManual )
      I_Contact( #iStep )
      I_Contact( #iModeSelectType )
      wire#w4
      Coil( #oAutoMode )
   END_RUNG
   RUNG wire#w1
      Contact( #iOneCycle )
   END_RUNG wire#w3
   RUNG wire#w1
      { S7_Templates := "SrcType := Int" } EQ_Contact(in1 := #iHMIModeSelect, in2 := 2)
      Contact( #iModeSelectType )
   END_RUNG wire#w4
   RUNG wire#w1
      { S7_Templates := "SrcType := Int" } EQ_Contact(in1 := #iHMIModeSelect, in2 := 4)
      Contact( #iModeSelectType )
   END_RUNG wire#w4
   RUNG wire#w1
      { S7_Templates := "SrcType := Int" } EQ_Contact(in1 := #iHMIModeSelect, in2 := 3)
      Contact( #iModeSelectType )
   END_RUNG wire#w4
   RUNG wire#w4
      { S7_GenerateENO := "TRUE" } Move(in := 2, out1 => #oMode)
   END_RUNG
   RUNG wire#w4
      { S7_Templates := "SrcType := Int" } EQ_Contact(in1 := #iHMIModeSelect, in2 := 4)
      Contact( #iModeSelectType )
      wire#w5
      { S7_GenerateENO := "TRUE" } Move(in := 4, out1 => #oMode)
      Coil( #oOneCycleMode )
   END_RUNG
   RUNG wire#w4
      Contact( #iOneCycle )
      I_Contact( #iModeSelectType )
   END_RUNG wire#w5
   RUNG wire#w1
      Contact( #iStep )
      I_Contact( #iAuto )
      I_Contact( #iManual )
      I_Contact( #iModeSelectType )
      wire#w6
      Coil( #oStepMode )
   END_RUNG
   RUNG wire#w1
      { S7_Templates := "SrcType := Int" } EQ_Contact(in1 := #iHMIModeSelect, in2 := 3)
      Contact( #iModeSelectType )
   END_RUNG wire#w6
   RUNG wire#w6
      { S7_GenerateENO := "TRUE" } Move(in := 3, out1 => #oMode)
   END_RUNG
   RUNG wire#w1
      Contact( #oEStopOK )
      Contact( #oControlON )
      Contact( #oMainPressureOK )
      wire#w7
      Contact( #oSafetyDoorOK )
      wire#w8
      { S7_Templates := "time_type := Time" } #sRunT.TON(pt := t#3s, et =>)
      wire#w9
      Coil( #oRun )
      Coil( #"oEnable alarm" )
   END_RUNG
   RUNG wire#w7
      Contact( #iSafetyByPass )
      Contact( #iManual )
   END_RUNG wire#w8
   RUNG wire#w9
      I_Contact( #tAlwaysOn )
      { S7_GenerateENO := "TRUE" } Move(in := 5, out1 => #oMode)
   END_RUNG
   // the same network as SCL:
   // ENO of a box is taken as its EN; it also drops when the box reports an error
   #oManualMode := #tAlwaysOn AND ((#iManual AND NOT #iAuto AND NOT #iStep AND NOT #iModeSelectType) OR ((#iHMIModeSelect = 1) AND #iModeSelectType));
   IF #oManualMode THEN #oMode := 1; END_IF;
   #oAutoMode := #tAlwaysOn AND (((#iAuto OR #iOneCycle) AND NOT #iManual AND NOT #iStep AND NOT #iModeSelectType) OR ((#iHMIModeSelect = 2) AND #iModeSelectType) OR ((#iHMIModeSelect = 4) AND #iModeSelectType) OR ((#iHMIModeSelect = 3) AND #iModeSelectType));
   IF #oAutoMode THEN #oMode := 2; END_IF;
   #_w1 := #oAutoMode AND (((#iHMIModeSelect = 4) AND #iModeSelectType) OR (#iOneCycle AND NOT #iModeSelectType));
   IF #_w1 THEN #oMode := 4; END_IF;
   #oOneCycleMode := #_w1;
   #oStepMode := #tAlwaysOn AND ((#iStep AND NOT #iAuto AND NOT #iManual AND NOT #iModeSelectType) OR ((#iHMIModeSelect = 3) AND #iModeSelectType));
   IF #oStepMode THEN #oMode := 3; END_IF;
   #sRunT(IN := #tAlwaysOn AND #oEStopOK AND #oControlON AND #oMainPressureOK AND (#oSafetyDoorOK OR (#iSafetyByPass AND #iManual)),   // TON
          PT := t#3s);
   #oRun := #sRunT.Q;
   #"oEnable alarm" := #sRunT.Q;
   IF #sRunT.Q AND NOT #tAlwaysOn THEN #oMode := 5; END_IF;
END_REGION

REGION Network 7: ChangeOverOK
   RUNG wire#powerrail
      Contact( #iChangeOverOK )
      { S7_Templates := "time_type := Time" } #sChangeOverTOF.TOF(pt := t#5S, et =>)
      Coil( #sChangeOverOK )
   END_RUNG
   // the same network as SCL:
   #sChangeOverTOF(IN := #iChangeOverOK, PT := t#5S);   // TOF
   #sChangeOverOK := #sChangeOverTOF.Q;
END_REGION

REGION Network 8: SystemReady
   RUNG wire#powerrail
      Contact( #oRun )
      Contact( #oAutoMode )
      Contact( #oMainPressureOK )
      Contact( #iFixtureOK )
      Contact( #sChangeOverOK )
      Contact( #iAllDeviceOK )
      Coil( #oReady )
   END_RUNG
   // the same network as SCL:
   #oReady := #oRun AND #oAutoMode AND #oMainPressureOK AND #iFixtureOK AND #sChangeOverOK AND #iAllDeviceOK;
END_REGION

REGION Network 9: SystemStatus
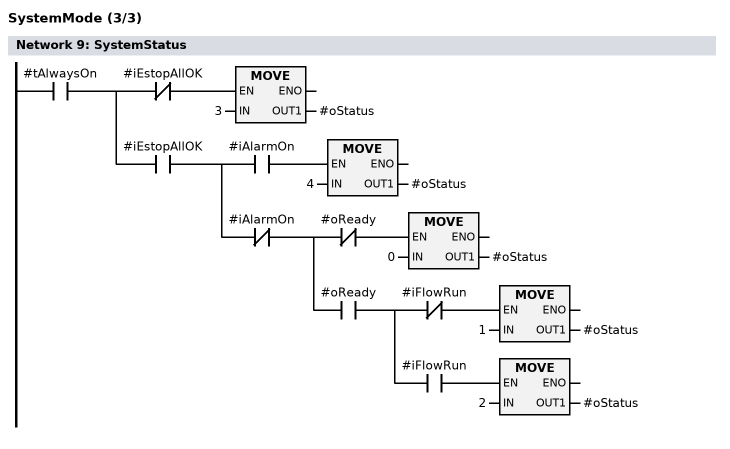
   RUNG wire#powerrail
      Contact( #tAlwaysOn )
      wire#w1
      I_Contact( #iEstopAllOK )
      Move(in := 3, out1 => #oStatus)
   END_RUNG
   RUNG wire#w1
      Contact( #iEstopAllOK )
      wire#w2
      Contact( #iAlarmOn )
      Move(in := 4, out1 => #oStatus)
   END_RUNG
   RUNG wire#w2
      I_Contact( #iAlarmOn )
      wire#w3
      I_Contact( #oReady )
      Move(in := 0, out1 => #oStatus)
   END_RUNG
   RUNG wire#w3
      Contact( #oReady )
      wire#w4
      I_Contact( #iFlowRun )
      Move(in := 1, out1 => #oStatus)
   END_RUNG
   RUNG wire#w4
      Contact( #iFlowRun )
      Move(in := 2, out1 => #oStatus)
   END_RUNG
   // the same network as SCL:
   IF #tAlwaysOn AND NOT #iEstopAllOK THEN #oStatus := 3; END_IF;
   #_w1 := #tAlwaysOn AND #iEstopAllOK;
   IF #_w1 AND #iAlarmOn THEN #oStatus := 4; END_IF;
   #_w2 := #_w1 AND NOT #iAlarmOn;
   IF #_w2 AND NOT #oReady THEN #oStatus := 0; END_IF;
   #_w3 := #_w2 AND #oReady;
   IF #_w3 AND NOT #iFlowRun THEN #oStatus := 1; END_IF;
   IF #_w3 AND #iFlowRun THEN #oStatus := 2; END_IF;
END_REGION
END_FUNCTION_BLOCK

FUNCTION_BLOCK "AutoProcessDataPopUp"   // FB1666, SCL
{ S7_Optimized_Access := 'TRUE' }
// stored: AutoNumber false, MemoryReserve 100, SetENOAutomatically false
   VAR_IN_OUT
      idx { ExternalAccessible := 'False'; ExternalVisible := 'False'; ExternalWritable := 'False'} : Int;
   END_VAR
   VAR_TEMP
      DefaultData : "ProcessDatad";
   END_VAR
BEGIN
   REGION read me
     // ============================================================================
     // PROGRAM START COMMENT
     // ============================================================================
     // EN:
     // FC_AutoProcessPopup handles popup visualization and editing of AutoProcess
     // data based on index from HMI.
     // The function provides:
     //  - automatic data loading from AutoProcessData according to selected index,
     //  - two-step confirmation for safe data overwrite (compare first, write second),
     //  - automatic reset of edit mode when index is changed,
     //  - delete functionality for selected record,
     //  - status bits for HMI to visualize pending changes and confirmation dialogs,
     //  - index range control (1..16).
     //
     // Data flow:
     // AutoProcessData  -> ActualSHowingData  (display mode)
     // ActualSHowingData -> AutoProcessData  (after double confirmation)
     //
     // Usage:
     // Call cyclically 
     // RMS index is taken from AutoProcess_HMI.IndexProcess.
     //
     // ----------------------------------------------------------------------------
     // CZ:
     // FC_AutoProcessPopup obsluhuje zobrazení a editaci dat AutoProcess podle
     // indexu z HMI.
     // Funkce zajišťuje:
     //  - automatické načítání dat z AutoProcessData podle zvoleného indexu,
     //  - dvoukrokové potvrzení zápisu (nejprve porovnání, poté zápis),
     //  - automatické zrušení editace při změně indexu,
     //  - mazání záznamu podle indexu,
     //  - stavové bity pro HMI (čekající změna, potvrzovací dialog),
     //  - kontrolu rozsahu indexu (1..16).
     //
     // Tok dat:
     // AutoProcessData  -> ActualSHowingData  (zobrazení)
     // ActualSHowingData -> AutoProcessData  (po potvrzení)
     //
     // Použití:
     // Volat cyklicky 
     // Index je čten z AutoProcess_HMI.IndexProcess.
     // ============================================================================

     // Statement section REGION

   END_REGION


   REGION IndexRangeCheck
     // EN: Clamp index to range 1..16
     // CZ: Oříznutí indexu do rozsahu 1..16
     IF #idx < 1 THEN
       #idx := 1;
       "AutoProcess_HMI".IndexProcess := #idx;
     ELSIF #idx > 16 THEN
       #idx := 16;
       "AutoProcess_HMI".IndexProcess := #idx;

     END_IF;
   END_REGION


   REGION IndexHandling
     // ---------------------------------------------------------------------------
     // EN: Detect index change and reset edit session
     // CZ: Detekce změny indexu a zrušení editace
     // ---------------------------------------------------------------------------
     #idx := "AutoProcess_HMI".IndexProcess;

     IF #idx <> "AutoProcess_HMI".Data_handling.LastIndex THEN
       "AutoProcess_HMI".Data_handling.UpdateData_switch := FALSE;
       "AutoProcess_HMI".Data_handling.UpdateData_Confirm := FALSE;
       "AutoProcess_HMI".Data_handling.FinalConfirm_Write := FALSE;
       "AutoProcess_HMI".Data_handling.ConfirmDialogActive := FALSE;
       "AutoProcess_HMI".Data_handling.ChangePending := FALSE;
       "AutoProcess_HMI".Data_handling.DeleteData := FALSE;
       "AutoProcess_HMI".Data_handling.LastIndex := #idx;
     END_IF;
   END_REGION



   REGION ShowData
     // ---------------------------------------------------------------------------
     // EN: Copy data to HMI if edit mode is inactive
     // CZ: Zobrazování dat – pokud není editace, kopíruj data z DB
     // ---------------------------------------------------------------------------
     IF NOT "AutoProcess_HMI".Data_handling.UpdateData_switch THEN
       CASE #idx OF
         1:
           "AutoProcess_HMI".ActualSHowingData := "AutoProcessData".A_ScanRotate;
         2:
           "AutoProcess_HMI".ActualSHowingData := "AutoProcessData".F_Robot1Grip1;
         3:
           "AutoProcess_HMI".ActualSHowingData := "AutoProcessData".F_Robot1Grip2;
         4:
           "AutoProcess_HMI".ActualSHowingData := "AutoProcessData".B_Press1;
         5:
           "AutoProcess_HMI".ActualSHowingData := "AutoProcessData".C_Glue;
         6:
           "AutoProcess_HMI".ActualSHowingData := "AutoProcessData".F_Robot2Grip1;
         7:
           "AutoProcess_HMI".ActualSHowingData := "AutoProcessData".F_Robot2Grip2;
         8:
           "AutoProcess_HMI".ActualSHowingData := "AutoProcessData".C_GlueNGBuffer;
         9:
           "AutoProcess_HMI".ActualSHowingData := "AutoProcessData".C_MagnScanNGBuffer;
         10:
           "AutoProcess_HMI".ActualSHowingData := "AutoProcessData".B_Press2;
         11:
           "AutoProcess_HMI".ActualSHowingData := "AutoProcessData".F_Robot3Grip1;
         12:
           "AutoProcess_HMI".ActualSHowingData := "AutoProcessData".F_Robot3Grip2;
         13:
           "AutoProcess_HMI".ActualSHowingData := "AutoProcessData".H_ShafeLine;
         14:
           "AutoProcess_HMI".ActualSHowingData := "AutoProcessData".J_MagnetBelt;
         15:
           "AutoProcess_HMI".ActualSHowingData := "AutoProcessData".K_ReserveBelt;
         16:
           "AutoProcess_HMI".ActualSHowingData := "AutoProcessData".L_UnloadBelt;
         ELSE
           ;
           // EN: invalid index / CZ: neplatný index
       END_CASE;
     END_IF;
   END_REGION



   REGION FirstConfirm
     // ---------------------------------------------------------------------------
     // EN: First confirmation → enable compare dialog
     // CZ: První potvrzení → aktivace porovnávacího dialogu
     // ---------------------------------------------------------------------------
     IF "AutoProcess_HMI".Data_handling.UpdateData_switch
       AND "AutoProcess_HMI".Data_handling.UpdateData_Confirm
       AND NOT "AutoProcess_HMI".Data_handling.ConfirmDialogActive THEN

       "AutoProcess_HMI".Data_handling.ConfirmDialogActive := TRUE;
       "AutoProcess_HMI".Data_handling.ChangePending := TRUE;

       "AutoProcess_HMI".Data_handling.UpdateData_Confirm := FALSE;
     END_IF;
   END_REGION



   REGION FinalWrite
     // ---------------------------------------------------------------------------
     // EN: Final confirmation → write to data DB
     // CZ: Finální potvrzení → zápis do DB
     // ---------------------------------------------------------------------------
     IF "AutoProcess_HMI".Data_handling.ConfirmDialogActive
       AND "AutoProcess_HMI".Data_handling.FinalConfirm_Write THEN

       CASE #idx OF
         1:
           "AutoProcessData".A_ScanRotate := "AutoProcess_HMI".ActualSHowingData;
         2:
           "AutoProcessData".F_Robot1Grip1 := "AutoProcess_HMI".ActualSHowingData;
         3:
           "AutoProcessData".F_Robot1Grip2 := "AutoProcess_HMI".ActualSHowingData;
         4:
           "AutoProcessData".B_Press1 := "AutoProcess_HMI".ActualSHowingData;
         5:
           "AutoProcessData".C_Glue := "AutoProcess_HMI".ActualSHowingData;
         6:
           "AutoProcessData".F_Robot2Grip1 := "AutoProcess_HMI".ActualSHowingData;
         7:
           "AutoProcessData".F_Robot2Grip2 := "AutoProcess_HMI".ActualSHowingData;
         8:
           "AutoProcessData".C_GlueNGBuffer := "AutoProcess_HMI".ActualSHowingData;
         9:
           "AutoProcessData".C_MagnScanNGBuffer := "AutoProcess_HMI".ActualSHowingData;
         10:
           "AutoProcessData".B_Press2 := "AutoProcess_HMI".ActualSHowingData;
         11:
           "AutoProcessData".F_Robot3Grip1 := "AutoProcess_HMI".ActualSHowingData;
         12:
           "AutoProcessData".F_Robot3Grip2 := "AutoProcess_HMI".ActualSHowingData;
         13:
           "AutoProcessData".H_ShafeLine := "AutoProcess_HMI".ActualSHowingData;
         14:
           "AutoProcessData".J_MagnetBelt := "AutoProcess_HMI".ActualSHowingData;
         15:
           "AutoProcessData".K_ReserveBelt := "AutoProcess_HMI".ActualSHowingData;
         16:
           "AutoProcessData".L_UnloadBelt := "AutoProcess_HMI".ActualSHowingData;
         ELSE
           ;
       END_CASE;

       // reset flags after write
       "AutoProcess_HMI".Data_handling.ConfirmDialogActive := FALSE;
       "AutoProcess_HMI".Data_handling.ChangePending := FALSE;
       "AutoProcess_HMI".Data_handling.FinalConfirm_Write := FALSE;
       "AutoProcess_HMI".Data_handling.UpdateData_switch := FALSE;
     END_IF;
   END_REGION



   REGION DeleteData
     // ---------------------------------------------------------------------------
     // EN: Delete selected Record (reset to default struct)
     // CZ: Smazání záznamu – vynulování struktury
     // ---------------------------------------------------------------------------
     IF "AutoProcess_HMI".Data_handling.DeleteData AND
       "AutoProcess_HMI".Data_handling.FinalConfirm_Write
       THEN

       CASE #idx OF
         1:
           "AutoProcessData".A_ScanRotate := #DefaultData;
         2:
           "AutoProcessData".F_Robot1Grip1 := #DefaultData;
         3:
           "AutoProcessData".F_Robot1Grip2 := #DefaultData;
         4:
           "AutoProcessData".B_Press1 := #DefaultData;
         5:
           "AutoProcessData".C_Glue := #DefaultData;
         6:
           "AutoProcessData".F_Robot2Grip1 := #DefaultData;
         7:
           "AutoProcessData".F_Robot2Grip2 := #DefaultData;
         8:
           "AutoProcessData".C_GlueNGBuffer := #DefaultData;
         9:
           "AutoProcessData".C_MagnScanNGBuffer := #DefaultData;
         10:
           "AutoProcessData".B_Press2 := #DefaultData;
         11:
           "AutoProcessData".F_Robot3Grip1 := #DefaultData;
         12:
           "AutoProcessData".F_Robot3Grip2 := #DefaultData;
         13:
           "AutoProcessData".H_ShafeLine := #DefaultData;
         14:
           "AutoProcessData".J_MagnetBelt := #DefaultData;
         15:
           "AutoProcessData".K_ReserveBelt := #DefaultData;
         16:
           "AutoProcessData".L_UnloadBelt := #DefaultData;
         ELSE
           ;
       END_CASE;

       // reset delete + editing states
       "AutoProcess_HMI".Data_handling.DeleteData := FALSE;
       "AutoProcess_HMI".Data_handling.UpdateData_switch := FALSE;
       "AutoProcess_HMI".Data_handling.UpdateData_Confirm := FALSE;
       "AutoProcess_HMI".Data_handling.FinalConfirm_Write := FALSE;
       "AutoProcess_HMI".Data_handling.ConfirmDialogActive := FALSE;
       "AutoProcess_HMI".Data_handling.ChangePending := FALSE;
     END_IF;
   END_REGION

   REGION StationProductIcons
     // EN: Set icon bits if station contains product (PartStatus <> 0)
     // CZ: Nastavení bitů ikony – stanice má kus, pokud PartStatus <> 0

     // 1 – A_ScanRotate
     "AutoProcess_HMI".StationHasProduct[1] :=
     "AutoProcessData".A_ScanRotate.PartStatus <> 0;

     // 2 – F_Robot1Grip1
     "AutoProcess_HMI".StationHasProduct[2] :=
     "AutoProcessData".F_Robot1Grip1.PartStatus <> 0;

     // 3 – F_Robot1Grip2
     "AutoProcess_HMI".StationHasProduct[3] :=
     "AutoProcessData".F_Robot1Grip2.PartStatus <> 0;

     // 4 – B_Press1
     "AutoProcess_HMI".StationHasProduct[4] :=
     "AutoProcessData".B_Press1.PartStatus <> 0;

     // 5 – C_Glue
     "AutoProcess_HMI".StationHasProduct[5] :=
     "AutoProcessData".C_Glue.PartStatus <> 0;

     // 6 – F_Robot2Grip1
     "AutoProcess_HMI".StationHasProduct[6] :=
     "AutoProcessData".F_Robot2Grip1.PartStatus <> 0;

     // 7 – F_Robot2Grip2
     "AutoProcess_HMI".StationHasProduct[7] :=
     "AutoProcessData".F_Robot2Grip2.PartStatus <> 0;

     // 8 – C_GlueNGBuffer
     "AutoProcess_HMI".StationHasProduct[8] :=
     "AutoProcessData".C_GlueNGBuffer.PartStatus <> 0;

     // 9 – C_MagnScanNGBuffer
     "AutoProcess_HMI".StationHasProduct[9] :=
     "AutoProcessData".C_MagnScanNGBuffer.PartStatus <> 0;

     // 10 – B_Press2
     "AutoProcess_HMI".StationHasProduct[10] :=
     "AutoProcessData".B_Press2.PartStatus <> 0;

     // 11 – F_Robot3Grip1
     "AutoProcess_HMI".StationHasProduct[11] :=
     "AutoProcessData".F_Robot3Grip1.PartStatus <> 0;

     // 12 – F_Robot3Grip2
     "AutoProcess_HMI".StationHasProduct[12] :=
     "AutoProcessData".F_Robot3Grip2.PartStatus <> 0;

     // 13 – H_ShafeLine
     "AutoProcess_HMI".StationHasProduct[13] :=
     "AutoProcessData".H_ShafeLine.PartStatus <> 0;

     // 14 – J_ShafeLine
     "AutoProcess_HMI".StationHasProduct[14] :=
     "AutoProcessData".J_MagnetBelt.PartStatus <> 0;

     // 15 – K_ShafeLine
     "AutoProcess_HMI".StationHasProduct[15] :=
     "AutoProcessData".K_ReserveBelt.PartStatus <> 0;

     // 16 – L_ShafeLine
     "AutoProcess_HMI".StationHasProduct[16] :=
     "AutoProcessData".L_UnloadBelt.PartStatus <> 0;

   END_REGION
END_FUNCTION_BLOCK

FUNCTION_BLOCK "FB_MES_Monitoring"   // FB4, SCL
{ S7_Optimized_Access := 'TRUE' }
// stored: IsIECCheckEnabled true, MemoryReserve 100, SetENOAutomatically false
   VAR_INPUT
      Enable : Bool := TRUE;
      Reset : Bool := FALSE;
      HeartbeatTimeout_MES : Time := T#6s;
      HeartbeatTimeout_PLC : Time := T#6s;
      CheckInTimeout : Time := T#10s;
      CheckOutTimeout : Time := T#10s;
      StoveCheckInTimeout : Time := T#10s;
   END_VAR
   VAR_IN_OUT
      Diag : "UDT_MES_Monitoring";
   END_VAR
   VAR
      _hbMesValue : Bool;
      _hbPlcValue : Bool;
      _errCode : Array[1..8] of DInt;
      _errText : Array[1..8] of String[128];
      _actErrIdx : Array[1..8] of Int;
      _actErrCnt : Int;
      _actErrPos : Int;
      _errRotateEnable : Bool;
      _tErrRotate { S7_SetPoint := 'True'} : TON_TIME;
      _hbMesLast : Bool;
      _hbPlcLast : Bool;
      _tHbMes { S7_SetPoint := 'True'} : TON_TIME;
      _tHbPlc { S7_SetPoint := 'True'} : TON_TIME;
      _tCi { S7_SetPoint := 'True'} : Array[1..8] of TON_TIME;
      _tCo { S7_SetPoint := 'True'} : Array[1..8] of TON_TIME;
      _tStove { S7_SetPoint := 'True'} : TON_TIME;
      _ciDonePrev : Array[1..8] of Bool;
      _coDonePrev : Array[1..8] of Bool;
      _ciOkPrev : Array[1..8] of Bool;
      _ciNgPrev : Array[1..8] of Bool;
      _coOkPrev : Array[1..8] of Bool;
      _coNgPrev : Array[1..8] of Bool;
      _ciTimeoutLatched : Array[1..8] of Bool;
      _coTimeoutLatched : Array[1..8] of Bool;
      _spDonePrev : Array[1..8] of Bool;
      _spOkPrev : Array[1..8] of Bool;
      _spNgPrev : Array[1..8] of Bool;
      _lrDonePrev : Array[1..8] of Bool;
      _lrOkPrev : Array[1..8] of Bool;
      _lrNgPrev : Array[1..8] of Bool;
      _stoveOkPrev : Bool;
      _stoveTimeoutLatched : Bool;
      _i : Int;
      _ciReq : Array[1..8] of Bool;
      _ciOk : Array[1..8] of Bool;
      _ciNg : Array[1..8] of Bool;
      _ciDone : Array[1..8] of Bool;
      _coReq : Array[1..8] of Bool;
      _coOk : Array[1..8] of Bool;
      _coNg : Array[1..8] of Bool;
      _coDone : Array[1..8] of Bool;
      _spOk : Array[1..8] of Bool;
      _spNg : Array[1..8] of Bool;
      _spDone : Array[1..8] of Bool;
      _lrOk : Array[1..8] of Bool;
      _lrNg : Array[1..8] of Bool;
      _lrDone : Array[1..8] of Bool;
      _stoveReq : Bool;
      _stoveOk : Bool;
   END_VAR
BEGIN
   (*
   ===============================================================================
   BLOCK / PURPOSE
   ===============================================================================
   This code builds a MES diagnostics snapshot (#Diag) from PLC<->MES handshake DBs.
   It:
   - Mirrors key signals into #Diag.Header / #Diag.LastError / #Diag.Special / #Diag.Station[i]
   - Measures heartbeat "age" and timeout for MES and PLC heartbeats
   - Tracks per-station handshake counters (OK / NG / Done / Timeout) with edge detection
   - Latches "UnexpectedDone" if Done arrives without active request
   - Implements RESET to clear all counters/flags in #Diag
   ===============================================================================
   ASSUMPTIONS / NOTES
   ===============================================================================
   - #_tHbMes, #_tHbPlc, #_tStove and #_tCi[], #_tCo[] are IEC TON timers
   - #HeartbeatTimeout_MES / _PLC, #CheckInTimeout, #CheckOutTimeout, #StoveCheckInTimeout are TIME
   - Indexing: stations are 1..8
   - "ChickIn" naming in tags is preserved as-is (typo likely in original DB)
   ===============================================================================
   *)

   REGION "GUARD / ENABLE"
     IF NOT #Enable THEN
       RETURN;
     END_IF;
   END_REGION

   REGION "READ RAW SIGNALS FROM DBs (PLC<->MES + LAST ERROR)"
     #_hbMesValue := "MEStoPLC"."MES.HeartbeatSignal";
     #_hbPlcValue := "PLCtoMES"."PLC.Unload_HeartbeatSignal";

     // Unload error per station
     #_errCode[1] := "Station1UnLoadData"."MES.ErrorCode";
     #_errText[1] := "Station1UnLoadData"."MES.ErrorMsg";

     #_errCode[2] := "Station2UnLoadData"."MES.ErrorCode";
     #_errText[2] := "Station2UnLoadData"."MES.ErrorMsg";

     #_errCode[3] := "Station3UnLoadData"."MES.ErrorCode";
     #_errText[3] := "Station3UnLoadData"."MES.ErrorMsg";

     #_errCode[4] := "Station4UnLoadData"."MES.ErrorCode";
     #_errText[4] := "Station4UnLoadData"."MES.ErrorMsg";

     #_errCode[5] := "Station5UnLoadData"."MES.ErrorCode";
     #_errText[5] := "Station5UnLoadData"."MES.ErrorMsg";

     #_errCode[6] := "Station6UnLoadData"."MES.ErrorCode";
     #_errText[6] := "Station6UnLoadData"."MES.ErrorMsg";

     #_errCode[7] := "Station7UnLoadData"."MES.ErrorCode";
     #_errText[7] := "Station7UnLoadData"."MES.ErrorMsg";

     #_errCode[8] := "Station8UnLoadData"."MES.ErrorCode";
     #_errText[8] := "Station8UnLoadData"."MES.ErrorMsg";

     #_stoveReq := "PLCtoMES"."PLC.Load_StoveCheckIn";
     #_stoveOk := "MEStoPLC"."MES.Load_StoveCheckInOk";
   END_REGION


   REGION "MAP TO DIAG HEADER + LAST ERROR"
     #Diag.Header.Heartbeat_MES := #_hbMesValue;
     #Diag.Header.Heartbeat_PLC := #_hbPlcValue;

   END_REGION

   REGION "ACTIVE ERROR BUFFER + 3s ROTATE TO #Diag.LastError"
     // rebuild buffer each scan
     #_actErrCnt := 0;
     FOR #_i := 1 TO 8 DO
       // --- aktivni chyba kriterium ---
       IF (#_errCode[#_i] <> 0) THEN
         #_actErrCnt := #_actErrCnt + 1;
         #_actErrIdx[#_actErrCnt] := #_i;
       END_IF;
     END_FOR;

     // expose count to diag
     #Diag.LastError.ActCnt_Errors := #_actErrCnt;

     // keep pointer valid
     IF (#_actErrCnt = 0) THEN
       #_actErrPos := 1;
       #_errRotateEnable := FALSE;

       // when nothing active -> clear last error
       #Diag.LastError."Station Number" := 0;
       #Diag.LastError.Code := 0;
       #Diag.LastError.Text := '';
     ELSE
       IF (#_actErrPos < 1) OR (#_actErrPos > #_actErrCnt) THEN
         #_actErrPos := 1;
       END_IF;

       // start rotation timer if not running
       IF NOT #_errRotateEnable THEN
         #_errRotateEnable := TRUE;
       END_IF;

       // run 3s timer while enabled
       #_tErrRotate(IN := #_errRotateEnable,
                    PT := T#3S);

       // when 3s elapsed -> advance and force timer reset next scan
       IF #_tErrRotate.Q THEN
         #_errRotateEnable := FALSE;   // TON resets next scan (1-scan gap je OK)

         #_actErrPos := #_actErrPos + 1;
         IF #_actErrPos > #_actErrCnt THEN
           #_actErrPos := 1;
         END_IF;
       END_IF;

       // write currently selected active error to global LastError
       #_i := #_actErrIdx[#_actErrPos];   // reuse #_i jako index stanice (1..8)

       #Diag.LastError."Station Number" := #_i;
       #Diag.LastError.Code := #_errCode[#_i];

       // orez text do String[128] (kdyz DB ma delsi)
       #Diag.LastError.Text := LEFT(IN := #_errText[#_i], L := 128);
     END_IF;
   END_REGION

   REGION "HEARTBEAT SUPERVISION - MES -> PLC"
     // If heartbeat toggled since last scan => reset timer (forces ET back to 0)
     IF #_hbMesValue <> #_hbMesLast THEN
       #_hbMesLast := #_hbMesValue;
       #_tHbMes(IN := FALSE,
                PT := t#100ms);
     END_IF;

     // Run timer continuously; Q becomes TRUE after PT elapsed without heartbeat change
     #_tHbMes(IN := TRUE,
              PT := #HeartbeatTimeout_MES);

     #Diag.Header.MES_HeartbeatTimeout := #_tHbMes.Q;   // TRUE = timeout reached
     #Diag.Header.MES_HeartbeatAge := #_tHbMes.ET;  // elapsed since last toggle
     #Diag.Header.MES_Online := NOT #_tHbMes.Q;
   END_REGION


   REGION "HEARTBEAT SUPERVISION - PLC -> MES"
     // If heartbeat toggled => reset PLC heartbeat timer
     IF #_hbPlcValue <> #_hbPlcLast THEN
       #_hbPlcLast := #_hbPlcValue;
       #_tHbPlc(IN := FALSE,
                PT := t#100ms);
     END_IF;

     // Run timer continuously
     #_tHbPlc(IN := TRUE,
              PT := #HeartbeatTimeout_PLC);

     #Diag.Header.PLC_HeartbeatTimeout := #_tHbPlc.Q;
     #Diag.Header.PLC_HeartbeatAge := #_tHbPlc.ET;
   END_REGION


   REGION "BUILD HANDSHAKE ARRAYS (READ INPUTS ONCE) - CHECK-IN REQ/OK/NG/DONE"
     // Check-in request bits (PLC -> MES), one per station
     #_ciReq[1] := "PLCtoMES"."PLC.Load_Station1ChickInReq";
     #_ciReq[2] := "PLCtoMES"."PLC.Load_Station2ChickInReq";
     #_ciReq[3] := "PLCtoMES"."PLC.Load_Station3ChickInReq";
     #_ciReq[4] := "PLCtoMES"."PLC.Load_Station4ChickInReq";
     #_ciReq[5] := "PLCtoMES"."PLC.Load_Station5ChickInReq";
     #_ciReq[6] := "PLCtoMES"."PLC.Load_Station6ChickInReq";
     #_ciReq[7] := "PLCtoMES"."PLC.Load_Station7ChickInReq";
     #_ciReq[8] := "PLCtoMES"."PLC.Load_Station8ChickInReq";

     // Check-in result bits from MES (OK / NG / Done)
     #_ciOk[1] := "MEStoPLC"."MES.Load_Station1PartOK";
     #_ciOk[2] := "MEStoPLC"."MES.Load_Station2PartOK";
     #_ciOk[3] := "MEStoPLC"."MES.Load_Station3PartOK";
     #_ciOk[4] := "MEStoPLC"."MES.Load_Station4PartOK";
     #_ciOk[5] := "MEStoPLC"."MES.Load_Station5PartOK";
     #_ciOk[6] := "MEStoPLC"."MES.Load_Station6PartOK";
     #_ciOk[7] := "MEStoPLC"."MES.Load_Station7PartOK";
     #_ciOk[8] := "MEStoPLC"."MES.Load_Station8PartOK";

     #_ciNg[1] := "MEStoPLC"."MES.Load_Station1PartNG";
     #_ciNg[2] := "MEStoPLC"."MES.Load_Station2PartNG";
     #_ciNg[3] := "MEStoPLC"."MES.Load_Station3PartNG";
     #_ciNg[4] := "MEStoPLC"."MES.Load_Station4PartNG";
     #_ciNg[5] := "MEStoPLC"."MES.Load_Station5PartNG";
     #_ciNg[6] := "MEStoPLC"."MES.Load_Station6PartNG";
     #_ciNg[7] := "MEStoPLC"."MES.Load_Station7PartNG";
     #_ciNg[8] := "MEStoPLC"."MES.Load_Station8PartNG";

     #_ciDone[1] := "MEStoPLC"."MES.Load_Station1ReqMesDone";
     #_ciDone[2] := "MEStoPLC"."MES.Load_Station2ReqMesDone";
     #_ciDone[3] := "MEStoPLC"."MES.Load_Station3ReqMesDone";
     #_ciDone[4] := "MEStoPLC"."MES.Load_Station4ReqMesDone";
     #_ciDone[5] := "MEStoPLC"."MES.Load_Station5ReqMesDone";
     #_ciDone[6] := "MEStoPLC"."MES.Load_Station6ReqMesDone";
     #_ciDone[7] := "MEStoPLC"."MES.Load_Station7ReqMesDone";
     #_ciDone[8] := "MEStoPLC"."MES.Load_Station8ReqMesDone";
   END_REGION


   REGION "BUILD HANDSHAKE ARRAYS (READ INPUTS ONCE) - CHECK-OUT REQ/OK/NG/DONE"
     // Check-out request bits (PLC -> MES): request to save unload data
     #_coReq[1] := "PLCtoMES"."PLC.Unload_Station1DataSaveReq";
     #_coReq[2] := "PLCtoMES"."PLC.Unload_Station2DataSaveReq";
     #_coReq[3] := "PLCtoMES"."PLC.Unload_Station3DataSaveReq";
     #_coReq[4] := "PLCtoMES"."PLC.Unload_Station4DataSaveReq";
     #_coReq[5] := "PLCtoMES"."PLC.Unload_Station5DataSaveReq";
     #_coReq[6] := "PLCtoMES"."PLC.Unload_Station6DataSaveReq";
     #_coReq[7] := "PLCtoMES"."PLC.Unload_Station7DataSaveReq";
     #_coReq[8] := "PLCtoMES"."PLC.Unload_Station8DataSaveReq";

     // Check-out results (OK/NG/Done) from MES
     #_coOk[1] := "MEStoPLC"."MES.Unload_ResultsStored1OK";
     #_coOk[2] := "MEStoPLC"."MES.Unload_ResultsStored2OK";
     #_coOk[3] := "MEStoPLC"."MES.Unload_ResultsStored3OK";
     #_coOk[4] := "MEStoPLC"."MES.Unload_ResultsStored4OK";
     #_coOk[5] := "MEStoPLC"."MES.Unload_ResultsStored5OK";
     #_coOk[6] := "MEStoPLC"."MES.Unload_ResultsStored6OK";
     #_coOk[7] := "MEStoPLC"."MES.Unload_ResultsStored7OK";
     #_coOk[8] := "MEStoPLC"."MES.Unload_ResultsStored8OK";

     #_coNg[1] := "MEStoPLC"."MES.Unload_ResultsStored1NG";
     #_coNg[2] := "MEStoPLC"."MES.Unload_ResultsStored2NG";
     #_coNg[3] := "MEStoPLC"."MES.Unload_ResultsStored3NG";
     #_coNg[4] := "MEStoPLC"."MES.Unload_ResultsStored4NG";
     #_coNg[5] := "MEStoPLC"."MES.Unload_ResultsStored5NG";
     #_coNg[6] := "MEStoPLC"."MES.Unload_ResultsStored6NG";
     #_coNg[7] := "MEStoPLC"."MES.Unload_ResultsStored7NG";
     #_coNg[8] := "MEStoPLC"."MES.Unload_ResultsStored8NG";

     #_coDone[1] := "MEStoPLC"."MES.Unload_ResultsStored1ReqMesDone";
     #_coDone[2] := "MEStoPLC"."MES.Unload_ResultsStored2ReqMesDone";
     #_coDone[3] := "MEStoPLC"."MES.Unload_ResultsStored3ReqMesDone";
     #_coDone[4] := "MEStoPLC"."MES.Unload_ResultsStored4ReqMesDone";
     #_coDone[5] := "MEStoPLC"."MES.Unload_ResultsStored5ReqMesDone";
     #_coDone[6] := "MEStoPLC"."MES.Unload_ResultsStored6ReqMesDone";
     #_coDone[7] := "MEStoPLC"."MES.Unload_ResultsStored7ReqMesDone";
     #_coDone[8] := "MEStoPLC"."MES.Unload_ResultsStored8ReqMesDone";
   END_REGION


   REGION "BUILD HANDSHAKE ARRAYS - SUBPART OK/NG/DONE (LOAD SIDE)"
     #_spOk[1] := "MEStoPLC"."MES.Load_SubPart1OK";
     #_spOk[2] := "MEStoPLC"."MES.Load_SubPart2OK";
     #_spOk[3] := "MEStoPLC"."MES.Load_SubPart3OK";
     #_spOk[4] := "MEStoPLC"."MES.Load_SubPart4OK";
     #_spOk[5] := "MEStoPLC"."MES.Load_SubPart5OK";
     #_spOk[6] := "MEStoPLC"."MES.Load_SubPart6OK";
     #_spOk[7] := "MEStoPLC"."MES.Load_SubPart7OK";
     #_spOk[8] := "MEStoPLC"."MES.Load_SubPart8OK";

     // NOTE: tags contain "...SubPartXtNG" (typo) - preserved exactly as given
     #_spNg[1] := "MEStoPLC"."MES.Load_SubPart1tNG";
     #_spNg[2] := "MEStoPLC"."MES.Load_SubPart2tNG";
     #_spNg[3] := "MEStoPLC"."MES.Load_SubPart3tNG";
     #_spNg[4] := "MEStoPLC"."MES.Load_SubPart4tNG";
     #_spNg[5] := "MEStoPLC"."MES.Load_SubPart5tNG";
     #_spNg[6] := "MEStoPLC"."MES.Load_SubPart6tNG";
     #_spNg[7] := "MEStoPLC"."MES.Load_SubPart7tNG";
     #_spNg[8] := "MEStoPLC"."MES.Load_SubPart8tNG";

     #_spDone[1] := "MEStoPLC"."MES.Load_SubPart1ReqMesDone";
     #_spDone[2] := "MEStoPLC"."MES.Load_SubPart2ReqMesDone";
     #_spDone[3] := "MEStoPLC"."MES.Load_SubPart3ReqMesDone";
     #_spDone[4] := "MEStoPLC"."MES.Load_SubPart4ReqMesDone";
     #_spDone[5] := "MEStoPLC"."MES.Load_SubPart5ReqMesDone";
     #_spDone[6] := "MEStoPLC"."MES.Load_SubPart6ReqMesDone";
     #_spDone[7] := "MEStoPLC"."MES.Load_SubPart7ReqMesDone";
     #_spDone[8] := "MEStoPLC"."MES.Load_SubPart8ReqMesDone";
   END_REGION


   REGION "BUILD HANDSHAKE ARRAYS - LOAD RESULTS STORED OK/NG/DONE (LOAD SIDE)"
     #_lrOk[1] := "MEStoPLC"."MES.Load_ResultsStored1OK";
     #_lrOk[2] := "MEStoPLC"."MES.Load_ResultsStored2OK";
     #_lrOk[3] := "MEStoPLC"."MES.Load_ResultsStored3OK";
     #_lrOk[4] := "MEStoPLC"."MES.Load_ResultsStored4OK";
     #_lrOk[5] := "MEStoPLC"."MES.Load_ResultsStored5OK";
     #_lrOk[6] := "MEStoPLC"."MES.Load_ResultsStored6OK";
     #_lrOk[7] := "MEStoPLC"."MES.Load_ResultsStored7OK";
     #_lrOk[8] := "MEStoPLC"."MES.Load_ResultsStored8OK";

     #_lrNg[1] := "MEStoPLC"."MES.Load_ResultsStored1NG";
     #_lrNg[2] := "MEStoPLC"."MES.Load_ResultsStored2NG";
     #_lrNg[3] := "MEStoPLC"."MES.Load_ResultsStored3NG";
     #_lrNg[4] := "MEStoPLC"."MES.Load_ResultsStored4NG";
     #_lrNg[5] := "MEStoPLC"."MES.Load_ResultsStored5NG";
     #_lrNg[6] := "MEStoPLC"."MES.Load_ResultsStored6NG";
     #_lrNg[7] := "MEStoPLC"."MES.Load_ResultsStored7NG";
     #_lrNg[8] := "MEStoPLC"."MES.Load_ResultsStored8NG";

     #_lrDone[1] := "MEStoPLC"."MES.Load_ResultsStored1ReqMesDone";
     #_lrDone[2] := "MEStoPLC"."MES.Load_ResultsStored2ReqMesDone";
     #_lrDone[3] := "MEStoPLC"."MES.Load_ResultsStored3ReqMesDone";
     #_lrDone[4] := "MEStoPLC"."MES.Load_ResultsStored4ReqMesDone";
     #_lrDone[5] := "MEStoPLC"."MES.Load_ResultsStored5ReqMesDone";
     #_lrDone[6] := "MEStoPLC"."MES.Load_ResultsStored6ReqMesDone";
     #_lrDone[7] := "MEStoPLC"."MES.Load_ResultsStored7ReqMesDone";
     #_lrDone[8] := "MEStoPLC"."MES.Load_ResultsStored8ReqMesDone";
   END_REGION


   REGION "RESET DIAGNOSTICS (COUNTERS + LATCHES)"
     IF #Reset THEN
       FOR #_i := 1 TO 8 DO
         // Station-level latches
         #Diag.Station[#_i].CheckIn.UnexpectedDone := FALSE;
         #Diag.Station[#_i].CheckOut.UnexpectedDone := FALSE;

         // Per-station counters: SubPart
         #Diag.Station[#_i].SubPart.CountOK := 0;
         #Diag.Station[#_i].SubPart.CountNG := 0;
         #Diag.Station[#_i].SubPart.CountDone := 0;

         // Per-station counters: LoadResultsStored
         #Diag.Station[#_i].LoadResultsStored.CountOK := 0;
         #Diag.Station[#_i].LoadResultsStored.CountNG := 0;
         #Diag.Station[#_i].LoadResultsStored.CountDone := 0;

         // Per-station counters: CheckIn
         #Diag.Station[#_i].CheckIn.CountOK := 0;
         #Diag.Station[#_i].CheckIn.CountNG := 0;
         #Diag.Station[#_i].CheckIn.CountDone := 0;
         #Diag.Station[#_i].CheckIn.CountTimeout := 0;

         // Per-station counters: CheckOut
         #Diag.Station[#_i].CheckOut.CountOK := 0;
         #Diag.Station[#_i].CheckOut.CountNG := 0;
         #Diag.Station[#_i].CheckOut.CountDone := 0;
         #Diag.Station[#_i].CheckOut.CountTimeout := 0;

         // Internal timeout latch states (avoid re-counting while timeout stays TRUE)
         #_ciTimeoutLatched[#_i] := FALSE;
         #_coTimeoutLatched[#_i] := FALSE;
       END_FOR;

       // Special (stove) counters / latches
       #Diag.Special.CountOk := 0;
       #Diag.Special.CountTimeout := 0;
       #_stoveTimeoutLatched := FALSE;
     END_IF;
   END_REGION


   REGION "RESET TOTAL COUNTERS (RE-CALCULATED EACH SCAN)"
     #Diag.Counters.TotalDone_CheckIn := 0;
     #Diag.Counters.TotalDone_CheckOut := 0;
     #Diag.Counters.TotalTimeout_CheckIn := 0;
     #Diag.Counters.TotalTimeout_CheckOut := 0;
     #Diag.Counters.TotalOK_CheckIn := 0;
     #Diag.Counters.TotalNG_CheckIn := 0;
     #Diag.Counters.TotalOK_CheckOut := 0;
     #Diag.Counters.TotalNG_CheckOut := 0;
   END_REGION


   REGION "MAIN LOOP 1..8 - STATION DIAGNOSTICS + EDGE COUNTERS + TIMEOUTS"
     FOR #_i := 1 TO 8 DO


       REGION "MAP STATION DATA (LOAD/UNLOAD) -> Diag.Station[i].*.DATA"
         // konstanta cisla stanice do Diag (pokud mas v UDT StationNumber)

         CASE #_i OF

           1:
             // ================== LOAD: Station1LoadData ==================
             #Diag.Station[#_i].CheckIn.DATA.PLC_PartTypeID := "Station1LoadData"."PLC.PartTypeID";
             #Diag.Station[#_i].CheckIn.DATA.PLC_StationRecipeNo := "Station1LoadData"."PLC.Station1RecipeNo";
             #Diag.Station[#_i].CheckIn.DATA.PLC_StationDMXCode := "Station1LoadData"."PLC.Station1DMXCode";
             #Diag.Station[#_i].CheckIn.DATA.PLC_StationStatus := "Station1LoadData"."PLC.StationStatus";
             #Diag.Station[#_i].CheckIn.DATA.MES_ErrorCode := "Station1LoadData"."MES.ErrorCode";
             #Diag.Station[#_i].CheckIn.DATA.MES_StatusBits := "Station1LoadData"."MES.StatusBits";
             #Diag.Station[#_i].CheckIn.DATA.MES_Cycle_ID := "Station1LoadData"."MES.Cycle_ID";
             #Diag.Station[#_i].CheckIn.DATA.MES_Unit_ParttypeID := "Station1LoadData"."MES.Unit_ParttypeID";

             // ================== UNLOAD: Station1UnLoadData ==================
             #Diag.Station[#_i].CheckOut.DATA.PLC_PartTypeID := "Station1UnLoadData"."PLC.PartTypeID";
             #Diag.Station[#_i].CheckOut.DATA.PLC_StationDMXCode := "Station1UnLoadData"."PLC.Station1DMXCode";
             #Diag.Station[#_i].CheckOut.DATA.PLC_StationRecipeNo := "Station1UnLoadData"."PLC.Station1RecipeNo";
             #Diag.Station[#_i].CheckOut.DATA.PLC_PartStatus := "Station1UnLoadData"."PLC.PartStatus";
             #Diag.Station[#_i].CheckOut.DATA.PLC_SubPartSN1 := "Station1UnLoadData"."PLC.SubPartSN1";
             #Diag.Station[#_i].CheckOut.DATA.PLC_TransferTime := "Station1UnLoadData"."PLC.TransferTime";
           //  #Diag.Station[#_i].CheckOut.DATA."PLC.NGCode" := "Station1UnLoadData"."PLC.NGCode";
             #Diag.Station[#_i].CheckOut.DATA.MES_ErrorCode := "Station1UnLoadData"."MES.ErrorCode";
             #Diag.Station[#_i].CheckOut.DATA.MES_ErrorMsg := "Station1UnLoadData"."MES.ErrorMsg";

           2:
             #Diag.Station[#_i].CheckIn.DATA.PLC_PartTypeID := "Station2LoadData"."PLC.PartTypeID";
             #Diag.Station[#_i].CheckIn.DATA.PLC_StationRecipeNo := "Station2LoadData"."PLC.Station2RecipeNo";
             #Diag.Station[#_i].CheckIn.DATA.PLC_StationDMXCode := "Station2LoadData"."PLC.Station2DMXCode";
          //   #Diag.Station[#_i].CheckIn.DATA."PLC.StationStatus" := "Station2LoadData"."PLC.StationStatus";
             #Diag.Station[#_i].CheckIn.DATA.MES_ErrorCode := "Station2LoadData"."MES.ErrorCode";
             #Diag.Station[#_i].CheckIn.DATA.MES_StatusBits := "Station2LoadData"."MES.StatusBits";
             #Diag.Station[#_i].CheckIn.DATA.MES_Cycle_ID := "Station2LoadData"."MES.Cycle_ID";
             #Diag.Station[#_i].CheckIn.DATA.MES_Unit_ParttypeID := "Station2LoadData"."MES.Unit_ParttypeID";

             #Diag.Station[#_i].CheckOut.DATA.PLC_PartTypeID := "Station2UnLoadData"."PLC.PartTypeID";
             #Diag.Station[#_i].CheckOut.DATA.PLC_StationDMXCode := "Station2UnLoadData"."PLC.Station2DMXCode";
             #Diag.Station[#_i].CheckOut.DATA.PLC_StationRecipeNo := "Station2UnLoadData"."PLC.Station2RecipeNo";
             #Diag.Station[#_i].CheckOut.DATA.PLC_PartStatus := "Station2UnLoadData"."PLC.PartStatus";
             #Diag.Station[#_i].CheckOut.DATA.PLC_SubPartSN1 := "Station2UnLoadData"."PLC.SubPartSN1";
             #Diag.Station[#_i].CheckOut.DATA.PLC_TransferTime := "Station2UnLoadData"."PLC.TransferTime";
         //    #Diag.Station[#_i].CheckOut.DATA."PLC.NGCode" := "Station2UnLoadData"."PLC.NGCode";
             #Diag.Station[#_i].CheckOut.DATA.MES_ErrorCode := "Station2UnLoadData"."MES.ErrorCode";
             #Diag.Station[#_i].CheckOut.DATA.MES_ErrorMsg := "Station2UnLoadData"."MES.ErrorMsg";

           3:
             #Diag.Station[#_i].CheckIn.DATA.PLC_PartTypeID := "Station3LoadData"."PLC.PartTypeID";
             #Diag.Station[#_i].CheckIn.DATA.PLC_StationRecipeNo := "Station3LoadData"."PLC.Station3RecipeNo";
             #Diag.Station[#_i].CheckIn.DATA.PLC_StationDMXCode := "Station3LoadData"."PLC.Station3DMXCode";
         //    #Diag.Station[#_i].CheckIn.DATA."PLC.StationStatus" := "Station3LoadData"."PLC.StationStatus";
             #Diag.Station[#_i].CheckIn.DATA.MES_ErrorCode := "Station3LoadData"."MES.ErrorCode";
             #Diag.Station[#_i].CheckIn.DATA.MES_StatusBits := "Station3LoadData"."MES.StatusBits";
             #Diag.Station[#_i].CheckIn.DATA.MES_Cycle_ID := "Station3LoadData"."MES.Cycle_ID";
             #Diag.Station[#_i].CheckIn.DATA.MES_Unit_ParttypeID := "Station3LoadData"."MES.Unit_ParttypeID";

             #Diag.Station[#_i].CheckOut.DATA.PLC_PartTypeID := "Station3UnLoadData"."PLC.PartTypeID";
             #Diag.Station[#_i].CheckOut.DATA.PLC_StationDMXCode := "Station3UnLoadData"."PLC.Station3DMXCode";
             #Diag.Station[#_i].CheckOut.DATA.PLC_StationRecipeNo := "Station3UnLoadData"."PLC.Station3RecipeNo";
             #Diag.Station[#_i].CheckOut.DATA.PLC_PartStatus := "Station3UnLoadData"."PLC.PartStatus";
             #Diag.Station[#_i].CheckOut.DATA.PLC_SubPartSN1 := "Station3UnLoadData"."PLC.SubPartSN1";
             #Diag.Station[#_i].CheckOut.DATA.PLC_TransferTime := "Station3UnLoadData"."PLC.TransferTime";
             #Diag.Station[#_i].CheckOut.DATA.PLC_NGCode := "Station3UnLoadData"."PLC.NGCode";
             #Diag.Station[#_i].CheckOut.DATA.MES_ErrorCode := "Station3UnLoadData"."MES.ErrorCode";
             #Diag.Station[#_i].CheckOut.DATA.MES_ErrorMsg := "Station3UnLoadData"."MES.ErrorMsg";

           4:
             #Diag.Station[#_i].CheckIn.DATA.PLC_PartTypeID := "Station4LoadData"."PLC.PartTypeID";
             #Diag.Station[#_i].CheckIn.DATA.PLC_StationRecipeNo := "Station4LoadData"."PLC.Station4RecipeNo";
             #Diag.Station[#_i].CheckIn.DATA.PLC_StationDMXCode := "Station4LoadData"."PLC.Station4DMXCode";
           //  #Diag.Station[#_i].CheckIn.DATA."PLC.StationStatus" := "Station4LoadData"."PLC.StationStatus";
             #Diag.Station[#_i].CheckIn.DATA.MES_ErrorCode := "Station4LoadData"."MES.ErrorCode";
             #Diag.Station[#_i].CheckIn.DATA.MES_StatusBits := "Station4LoadData"."MES.StatusBits";
             #Diag.Station[#_i].CheckIn.DATA.MES_Cycle_ID := "Station4LoadData"."MES.Cycle_ID";
             #Diag.Station[#_i].CheckIn.DATA.MES_Unit_ParttypeID := "Station4LoadData"."MES.Unit_ParttypeID";

             #Diag.Station[#_i].CheckOut.DATA.PLC_PartTypeID := "Station4UnLoadData"."PLC.PartTypeID";
             #Diag.Station[#_i].CheckOut.DATA.PLC_StationDMXCode := "Station4UnLoadData"."PLC.Station4DMXCode";
             #Diag.Station[#_i].CheckOut.DATA.PLC_StationRecipeNo := "Station4UnLoadData"."PLC.Station4RecipeNo";
             #Diag.Station[#_i].CheckOut.DATA.PLC_PartStatus := "Station4UnLoadData"."PLC.PartStatus";
             #Diag.Station[#_i].CheckOut.DATA.PLC_SubPartSN1 := "Station4UnLoadData"."PLC.SubPartSN1";
             #Diag.Station[#_i].CheckOut.DATA.PLC_TransferTime := "Station4UnLoadData"."PLC.TransferTime";
         //    #Diag.Station[#_i].CheckOut.DATA."PLC.NGCode" := "Station4UnLoadData"."PLC.NGCode";
             #Diag.Station[#_i].CheckOut.DATA.MES_ErrorCode := "Station4UnLoadData"."MES.ErrorCode";
             #Diag.Station[#_i].CheckOut.DATA.MES_ErrorMsg := "Station4UnLoadData"."MES.ErrorMsg";

           5:
             #Diag.Station[#_i].CheckIn.DATA.PLC_PartTypeID := "Station5LoadData"."PLC.PartTypeID";
             #Diag.Station[#_i].CheckIn.DATA.PLC_StationRecipeNo := "Station5LoadData"."PLC.Station5RecipeNo";
             #Diag.Station[#_i].CheckIn.DATA.PLC_StationDMXCode := "Station5LoadData"."PLC.Station5DMXCode";
        //     #Diag.Station[#_i].CheckIn.DATA."PLC.StationStatus" := "Station5LoadData"."PLC.StationStatus";
             #Diag.Station[#_i].CheckIn.DATA.MES_ErrorCode := "Station5LoadData"."MES.ErrorCode";
             #Diag.Station[#_i].CheckIn.DATA.MES_StatusBits := "Station5LoadData"."MES.StatusBits";
             #Diag.Station[#_i].CheckIn.DATA.MES_Cycle_ID := "Station5LoadData"."MES.Cycle_ID";
             #Diag.Station[#_i].CheckIn.DATA.MES_Unit_ParttypeID := "Station5LoadData"."MES.Unit_ParttypeID";

             #Diag.Station[#_i].CheckOut.DATA.PLC_PartTypeID := "Station5UnLoadData"."PLC.PartTypeID";
             #Diag.Station[#_i].CheckOut.DATA.PLC_StationDMXCode := "Station5UnLoadData"."PLC.Station5DMXCode";
             #Diag.Station[#_i].CheckOut.DATA.PLC_StationRecipeNo := "Station5UnLoadData"."PLC.Station5RecipeNo";
             #Diag.Station[#_i].CheckOut.DATA.PLC_PartStatus := "Station5UnLoadData"."PLC.PartStatus";
             #Diag.Station[#_i].CheckOut.DATA.PLC_SubPartSN1 := "Station5UnLoadData"."PLC.SubPartSN1";
             #Diag.Station[#_i].CheckOut.DATA.PLC_TransferTime := "Station5UnLoadData"."PLC.TransferTime";
             #Diag.Station[#_i].CheckOut.DATA.PLC_NGCode := "Station5UnLoadData"."PLC.NGCode";
             #Diag.Station[#_i].CheckOut.DATA.MES_ErrorCode := "Station5UnLoadData"."MES.ErrorCode";
             #Diag.Station[#_i].CheckOut.DATA.MES_ErrorMsg := "Station5UnLoadData"."MES.ErrorMsg";

           6:
             #Diag.Station[#_i].CheckIn.DATA.PLC_PartTypeID := "Station6LoadData"."PLC.PartTypeID";
             #Diag.Station[#_i].CheckIn.DATA.PLC_StationRecipeNo := "Station6LoadData"."PLC.Station6RecipeNo";
             #Diag.Station[#_i].CheckIn.DATA.PLC_StationDMXCode := "Station6LoadData"."PLC.Station6DMXCode";
         //    #Diag.Station[#_i].CheckIn.DATA."PLC.StationStatus" := "Station6LoadData"."PLC.StationStatus";
             #Diag.Station[#_i].CheckIn.DATA.MES_ErrorCode := "Station6LoadData"."MES.ErrorCode";
             #Diag.Station[#_i].CheckIn.DATA.MES_StatusBits := "Station6LoadData"."MES.StatusBits";
             #Diag.Station[#_i].CheckIn.DATA.MES_Cycle_ID := "Station6LoadData"."MES.Cycle_ID";
             #Diag.Station[#_i].CheckIn.DATA.MES_Unit_ParttypeID := "Station6LoadData"."MES.Unit_ParttypeID";

             #Diag.Station[#_i].CheckOut.DATA.PLC_PartTypeID := "Station6UnLoadData"."PLC.PartTypeID";
             #Diag.Station[#_i].CheckOut.DATA.PLC_StationDMXCode := "Station6UnLoadData"."PLC.Station6DMXCode";
             #Diag.Station[#_i].CheckOut.DATA.PLC_StationRecipeNo := "Station6UnLoadData"."PLC.Station6RecipeNo";
             #Diag.Station[#_i].CheckOut.DATA.PLC_PartStatus := "Station6UnLoadData"."PLC.PartStatus";
             #Diag.Station[#_i].CheckOut.DATA.PLC_SubPartSN1 := "Station6UnLoadData"."PLC.SubPartSN1";
             #Diag.Station[#_i].CheckOut.DATA.PLC_TransferTime := "Station6UnLoadData"."PLC.TransferTime";
         //    #Diag.Station[#_i].CheckOut.DATA."PLC.NGCode" := "Station6UnLoadData"."PLC.NGCode";
             #Diag.Station[#_i].CheckOut.DATA.MES_ErrorCode := "Station6UnLoadData"."MES.ErrorCode";
             #Diag.Station[#_i].CheckOut.DATA.MES_ErrorMsg := "Station6UnLoadData"."MES.ErrorMsg";

           7:
             #Diag.Station[#_i].CheckIn.DATA.PLC_PartTypeID := "Station7LoadData"."PLC.PartTypeID";
             #Diag.Station[#_i].CheckIn.DATA.PLC_StationRecipeNo := "Station7LoadData"."PLC.Station7RecipeNo";
             #Diag.Station[#_i].CheckIn.DATA.PLC_StationDMXCode := "Station7LoadData"."PLC.Station7DMXCode";
     //        #Diag.Station[#_i].CheckIn.DATA."PLC.StationStatus" := "Station7LoadData"."PLC.StationStatus";
             #Diag.Station[#_i].CheckIn.DATA.MES_ErrorCode := "Station7LoadData"."MES.ErrorCode";
             #Diag.Station[#_i].CheckIn.DATA.MES_StatusBits := "Station7LoadData"."MES.StatusBits";
             #Diag.Station[#_i].CheckIn.DATA.MES_Cycle_ID := "Station7LoadData"."MES.Cycle_ID";
             #Diag.Station[#_i].CheckIn.DATA.MES_Unit_ParttypeID := "Station7LoadData"."MES.Unit_ParttypeID";

             #Diag.Station[#_i].CheckOut.DATA.PLC_PartTypeID := "Station7UnLoadData"."PLC.PartTypeID";
             #Diag.Station[#_i].CheckOut.DATA.PLC_StationDMXCode := "Station7UnLoadData"."PLC.Station7DMXCode";
             #Diag.Station[#_i].CheckOut.DATA.PLC_StationRecipeNo := "Station7UnLoadData"."PLC.Station7RecipeNo";
             #Diag.Station[#_i].CheckOut.DATA.PLC_PartStatus := "Station7UnLoadData"."PLC.PartStatus";
             #Diag.Station[#_i].CheckOut.DATA.PLC_SubPartSN1 := "Station7UnLoadData"."PLC.SubPartSN1";
             #Diag.Station[#_i].CheckOut.DATA.PLC_TransferTime := "Station7UnLoadData"."PLC.TransferTime";
             #Diag.Station[#_i].CheckOut.DATA.PLC_NGCode := "Station7UnLoadData"."PLC.NGCode";
             #Diag.Station[#_i].CheckOut.DATA.MES_ErrorCode := "Station7UnLoadData"."MES.ErrorCode";
             #Diag.Station[#_i].CheckOut.DATA.MES_ErrorMsg := "Station7UnLoadData"."MES.ErrorMsg";

           8:
             #Diag.Station[#_i].CheckIn.DATA.PLC_PartTypeID := "Station8LoadData"."PLC.PartTypeID";
             #Diag.Station[#_i].CheckIn.DATA.PLC_StationRecipeNo := "Station8LoadData"."PLC.Station8RecipeNo";
             #Diag.Station[#_i].CheckIn.DATA.PLC_StationDMXCode := "Station8LoadData"."PLC.Station8DMXCode";
   //          #Diag.Station[#_i].CheckIn.DATA."PLC.StationStatus" := "Station8LoadData"."PLC.StationStatus";
             #Diag.Station[#_i].CheckIn.DATA.MES_ErrorCode := "Station8LoadData"."MES.ErrorCode";
             #Diag.Station[#_i].CheckIn.DATA.MES_StatusBits := "Station8LoadData"."MES.StatusBits";
             #Diag.Station[#_i].CheckIn.DATA.MES_Cycle_ID := "Station8LoadData"."MES.Cycle_ID";
             #Diag.Station[#_i].CheckIn.DATA.MES_Unit_ParttypeID := "Station8LoadData"."MES.Unit_ParttypeID";

             #Diag.Station[#_i].CheckOut.DATA.PLC_PartTypeID := "Station8UnLoadData"."PLC.PartTypeID";
        //     #Diag.Station[#_i].CheckOut.DATA."PLC.StationDMXCode" := "Station8UnLoadData"."PLC.Station8DMXCode";
       //      #Diag.Station[#_i].CheckOut.DATA."PLC.StationRecipeNo" := "Station8UnLoadData"."PLC.Station8RecipeNo";
             #Diag.Station[#_i].CheckOut.DATA.PLC_PartStatus := "Station8UnLoadData"."PLC.PartStatus";
             #Diag.Station[#_i].CheckOut.DATA.PLC_SubPartSN1 := "Station8UnLoadData"."PLC.SubPartSN1";
             #Diag.Station[#_i].CheckOut.DATA.PLC_TransferTime := "Station8UnLoadData"."PLC.TransferTime";
       //      #Diag.Station[#_i].CheckOut.DATA."PLC.NGCode" := "Station8UnLoadData"."PLC.NGCode";
             #Diag.Station[#_i].CheckOut.DATA.MES_ErrorCode := "Station8UnLoadData"."MES.ErrorCode";
             #Diag.Station[#_i].CheckOut.DATA.MES_ErrorMsg := "Station8UnLoadData"."MES.ErrorMsg";

         END_CASE;
       END_REGION


       // --------------------------------------------------------------------------
       // CHECK-IN DIAG (Load)
       // --------------------------------------------------------------------------
       #Diag.Station[#_i].CheckIn.Req := #_ciReq[#_i];
       #Diag.Station[#_i].CheckIn.OK := #_ciOk[#_i];
       #Diag.Station[#_i].CheckIn.NG := #_ciNg[#_i];
       #Diag.Station[#_i].CheckIn.Done := #_ciDone[#_i];

       // Invalid state detector: OK and NG simultaneously
       #Diag.Station[#_i].CheckIn.BothOkNg := #_ciOk[#_i] AND #_ciNg[#_i];

       // Rising edge count: OK
       IF #_ciOk[#_i] AND (NOT #_ciOkPrev[#_i]) THEN
         #Diag.Station[#_i].CheckIn.CountOK := #Diag.Station[#_i].CheckIn.CountOK + 1;
       END_IF;
       #_ciOkPrev[#_i] := #_ciOk[#_i];

       // Rising edge count: NG
       IF #_ciNg[#_i] AND (NOT #_ciNgPrev[#_i]) THEN
         #Diag.Station[#_i].CheckIn.CountNG := #Diag.Station[#_i].CheckIn.CountNG + 1;
       END_IF;
       #_ciNgPrev[#_i] := #_ciNg[#_i];

       // Timer: measure duration of active request
       IF #_ciReq[#_i] THEN
         #_tCi[#_i](IN := TRUE,
                    PT := #CheckInTimeout);
         #Diag.Station[#_i].CheckIn.InProgress := TRUE;
       ELSE
         // Reset timer when request is inactive
         #_tCi[#_i](IN := FALSE,
                    PT := t#100ms);
         #Diag.Station[#_i].CheckIn.InProgress := FALSE;
       END_IF;

       #Diag.Station[#_i].CheckIn.Elapsed := #_tCi[#_i].ET;

       // Timeout: timer expired while request still active and Done not received
       #Diag.Station[#_i].CheckIn.Timeout :=
       #_tCi[#_i].Q AND #_ciReq[#_i] AND (NOT #_ciDone[#_i]);

       // Count timeout only on first scan of timeout assertion (latch)
       IF #Diag.Station[#_i].CheckIn.Timeout AND (NOT #_ciTimeoutLatched[#_i]) THEN
         #_ciTimeoutLatched[#_i] := TRUE;
         #Diag.Station[#_i].CheckIn.CountTimeout := #Diag.Station[#_i].CheckIn.CountTimeout + 1;
       END_IF;

       // Release latch when timeout condition clears
       IF NOT #Diag.Station[#_i].CheckIn.Timeout THEN
         #_ciTimeoutLatched[#_i] := FALSE;
       END_IF;

       // Rising edge count: Done + UnexpectedDone latch if no active request
       IF #_ciDone[#_i] AND (NOT #_ciDonePrev[#_i]) THEN
         #Diag.Station[#_i].CheckIn.CountDone := #Diag.Station[#_i].CheckIn.CountDone + 1;

         // Done without request: indicates inconsistent handshake timing or stale signals
         IF NOT #_ciReq[#_i] THEN
           #Diag.Station[#_i].CheckIn.UnexpectedDone := TRUE;
         END_IF;
       END_IF;
       #_ciDonePrev[#_i] := #_ciDone[#_i];

       // Add to totals (totals are sum of per-station counters)
       #Diag.Counters.TotalDone_CheckIn := #Diag.Counters.TotalDone_CheckIn + #Diag.Station[#_i].CheckIn.CountDone;
       #Diag.Counters.TotalTimeout_CheckIn := #Diag.Counters.TotalTimeout_CheckIn + #Diag.Station[#_i].CheckIn.CountTimeout;
       #Diag.Counters.TotalOK_CheckIn := #Diag.Counters.TotalOK_CheckIn + #Diag.Station[#_i].CheckIn.CountOK;
       #Diag.Counters.TotalNG_CheckIn := #Diag.Counters.TotalNG_CheckIn + #Diag.Station[#_i].CheckIn.CountNG;


       // --------------------------------------------------------------------------
       // CHECK-OUT DIAG (Unload)
       // --------------------------------------------------------------------------
       #Diag.Station[#_i].CheckOut.Req := #_coReq[#_i];
       #Diag.Station[#_i].CheckOut.StoredOK := #_coOk[#_i];
       #Diag.Station[#_i].CheckOut.StoredNG := #_coNg[#_i];
       #Diag.Station[#_i].CheckOut.Done := #_coDone[#_i];

       // Invalid state detector: OK and NG simultaneously
       #Diag.Station[#_i].CheckOut.BothOkNg := #_coOk[#_i] AND #_coNg[#_i];

       // Rising edge count: OK
       IF #_coOk[#_i] AND (NOT #_coOkPrev[#_i]) THEN
         #Diag.Station[#_i].CheckOut.CountOK := #Diag.Station[#_i].CheckOut.CountOK + 1;
       END_IF;
       #_coOkPrev[#_i] := #_coOk[#_i];

       // Rising edge count: NG
       IF #_coNg[#_i] AND (NOT #_coNgPrev[#_i]) THEN
         #Diag.Station[#_i].CheckOut.CountNG := #Diag.Station[#_i].CheckOut.CountNG + 1;
       END_IF;
       #_coNgPrev[#_i] := #_coNg[#_i];

       // Timer: measure duration of active request
       IF #_coReq[#_i] THEN
         #_tCo[#_i](IN := TRUE,
                    PT := #CheckOutTimeout);
         #Diag.Station[#_i].CheckOut.InProgress := TRUE;
       ELSE
         // Reset timer when request is inactive
         #_tCo[#_i](IN := FALSE,
                    PT := t#100ms);
         #Diag.Station[#_i].CheckOut.InProgress := FALSE;
       END_IF;

       #Diag.Station[#_i].CheckOut.Elapsed := #_tCo[#_i].ET;

       // Timeout: timer expired while request still active and Done not received
       #Diag.Station[#_i].CheckOut.Timeout :=
       #_tCo[#_i].Q AND #_coReq[#_i] AND (NOT #_coDone[#_i]);

       // Count timeout only once per timeout episode (latch)
       IF #Diag.Station[#_i].CheckOut.Timeout AND (NOT #_coTimeoutLatched[#_i]) THEN
         #_coTimeoutLatched[#_i] := TRUE;
         #Diag.Station[#_i].CheckOut.CountTimeout := #Diag.Station[#_i].CheckOut.CountTimeout + 1;
       END_IF;

       // Release latch when timeout clears
       IF NOT #Diag.Station[#_i].CheckOut.Timeout THEN
         #_coTimeoutLatched[#_i] := FALSE;
       END_IF;

       // Rising edge count: Done + UnexpectedDone latch if no active request
       IF #_coDone[#_i] AND (NOT #_coDonePrev[#_i]) THEN
         #Diag.Station[#_i].CheckOut.CountDone := #Diag.Station[#_i].CheckOut.CountDone + 1;

         // Done without request: indicates inconsistent handshake timing or stale signals
         IF NOT #_coReq[#_i] THEN
           #Diag.Station[#_i].CheckOut.UnexpectedDone := TRUE;
         END_IF;
       END_IF;
       #_coDonePrev[#_i] := #_coDone[#_i];

       // Add to totals
       #Diag.Counters.TotalDone_CheckOut := #Diag.Counters.TotalDone_CheckOut + #Diag.Station[#_i].CheckOut.CountDone;
       #Diag.Counters.TotalTimeout_CheckOut := #Diag.Counters.TotalTimeout_CheckOut + #Diag.Station[#_i].CheckOut.CountTimeout;
       #Diag.Counters.TotalOK_CheckOut := #Diag.Counters.TotalOK_CheckOut + #Diag.Station[#_i].CheckOut.CountOK;
       #Diag.Counters.TotalNG_CheckOut := #Diag.Counters.TotalNG_CheckOut + #Diag.Station[#_i].CheckOut.CountNG;


       // --------------------------------------------------------------------------
       // SUBPART DIAG (MES classification for subparts)
       // --------------------------------------------------------------------------
       #Diag.Station[#_i].SubPart.OK := #_spOk[#_i];
       #Diag.Station[#_i].SubPart.NG := #_spNg[#_i];
       #Diag.Station[#_i].SubPart.Done := #_spDone[#_i];

       #Diag.Station[#_i].SubPart.BothOkNg := #_spOk[#_i] AND #_spNg[#_i];

       // Rising edge count: OK
       IF #_spOk[#_i] AND (NOT #_spOkPrev[#_i]) THEN
         #Diag.Station[#_i].SubPart.CountOK := #Diag.Station[#_i].SubPart.CountOK + 1;
       END_IF;
       #_spOkPrev[#_i] := #_spOk[#_i];

       // Rising edge count: NG
       IF #_spNg[#_i] AND (NOT #_spNgPrev[#_i]) THEN
         #Diag.Station[#_i].SubPart.CountNG := #Diag.Station[#_i].SubPart.CountNG + 1;
       END_IF;
       #_spNgPrev[#_i] := #_spNg[#_i];

       // Rising edge count: Done
       IF #_spDone[#_i] AND (NOT #_spDonePrev[#_i]) THEN
         #Diag.Station[#_i].SubPart.CountDone := #Diag.Station[#_i].SubPart.CountDone + 1;
       END_IF;
       #_spDonePrev[#_i] := #_spDone[#_i];


       // --------------------------------------------------------------------------
       // LOAD RESULTS STORED DIAG (MES confirm storing results for load side)
       // --------------------------------------------------------------------------
       #Diag.Station[#_i].LoadResultsStored.OK := #_lrOk[#_i];
       #Diag.Station[#_i].LoadResultsStored.NG := #_lrNg[#_i];
       #Diag.Station[#_i].LoadResultsStored.Done := #_lrDone[#_i];

       #Diag.Station[#_i].LoadResultsStored.BothOkNg := #_lrOk[#_i] AND #_lrNg[#_i];

       // Rising edge count: OK
       IF #_lrOk[#_i] AND (NOT #_lrOkPrev[#_i]) THEN
         #Diag.Station[#_i].LoadResultsStored.CountOK := #Diag.Station[#_i].LoadResultsStored.CountOK + 1;
       END_IF;
       #_lrOkPrev[#_i] := #_lrOk[#_i];

       // Rising edge count: NG
       IF #_lrNg[#_i] AND (NOT #_lrNgPrev[#_i]) THEN
         #Diag.Station[#_i].LoadResultsStored.CountNG := #Diag.Station[#_i].LoadResultsStored.CountNG + 1;
       END_IF;
       #_lrNgPrev[#_i] := #_lrNg[#_i];

       // Rising edge count: Done
       IF #_lrDone[#_i] AND (NOT #_lrDonePrev[#_i]) THEN
         #Diag.Station[#_i].LoadResultsStored.CountDone := #Diag.Station[#_i].LoadResultsStored.CountDone + 1;
       END_IF;
       #_lrDonePrev[#_i] := #_lrDone[#_i];

     END_FOR;
   END_REGION


   REGION "SPECIAL HANDSHAKE - STOVE CHECK-IN (LOAD)"
     #Diag.Special.StoveCheckInReq := #_stoveReq;
     #Diag.Special.StoveCheckInOk := #_stoveOk;
     #Diag.Special.InProgress := #_stoveReq;

     // Timer runs while request active
     #_tStove(IN := #_stoveReq,
              PT := #StoveCheckInTimeout);

     #Diag.Special.Elapsed := #_tStove.ET;

     // Timeout: PT elapsed and still no OK
     #Diag.Special.Timeout := #_tStove.Q AND #_stoveReq AND (NOT #_stoveOk);

     // Rising edge count: OK
     IF #_stoveOk AND (NOT #_stoveOkPrev) THEN
       #Diag.Special.CountOk := #Diag.Special.CountOk + 1;
     END_IF;
     #_stoveOkPrev := #_stoveOk;

     // Count timeout only once per timeout episode
     IF #Diag.Special.Timeout AND (NOT #_stoveTimeoutLatched) THEN
       #_stoveTimeoutLatched := TRUE;
       #Diag.Special.CountTimeout := #Diag.Special.CountTimeout + 1;
     END_IF;

     IF NOT #Diag.Special.Timeout THEN
       #_stoveTimeoutLatched := FALSE;
     END_IF;
   END_REGION
END_FUNCTION_BLOCK

FUNCTION "FC_Teach_Recipe_Transfer" : Void   // FC4, SCL
{ S7_Optimized_Access := 'TRUE' }
// stored: SetENOAutomatically false
   VAR_IN_OUT
      recipeIndex : USInt;
   END_VAR
BEGIN

   // Clamp recipe index to array bounds [1..10].
   // 
   IF #recipeIndex< 1 THEN
     #recipeIndex := 1;
   ELSIF #recipeIndex> 10 THEN
     #recipeIndex := 10;
   END_IF;

   // Block read/save if teach mode is not active.
   IF NOT "DB_PARAMETERS_TEACH".HMI_PAGE_CONTROL.TEACH_MODE_ACTIVE THEN
     "DB_PARAMETERS_TEACH".HMI_PAGE_CONTROL.READ_CHOOSED_RECIPE := FALSE;
     "DB_PARAMETERS_TEACH".HMI_PAGE_CONTROL.SAVE_CHANGES_IN_RECIPE := FALSE;
     RETURN;
   END_IF;

   // Read selected recipe into teach screen values.
   IF "DB_PARAMETERS_TEACH".HMI_PAGE_CONTROL.READ_CHOOSED_RECIPE THEN
     "DB_PARAMETERS_TEACH"."TEACH SCREEN VALUES" :=
     "DB_ALL_PROCESS_PARAMETERS".PRODUCT_TYPE[#recipeIndex];
    // "DB_ALL_PROCESS_PARAMETERS".ACTUAL_CHOOSEN_TYPE :=
   //  "DB_ALL_PROCESS_PARAMETERS".PRODUCT_TYPE[#recipeIndex];
     "DB_PARAMETERS_TEACH".HMI_PAGE_CONTROL.READ_CHOOSED_RECIPE := FALSE;
   END_IF;

   // Save teach screen values back into selected recipe.
    IF "DB_PARAMETERS_TEACH".HMI_PAGE_CONTROL.SAVE_CHANGES_IN_RECIPE THEN
     "DB_ALL_PROCESS_PARAMETERS".PRODUCT_TYPE[#recipeIndex] :=
     "DB_PARAMETERS_TEACH"."TEACH SCREEN VALUES";
    // "DB_ALL_PROCESS_PARAMETERS".ACTUAL_CHOOSEN_TYPE :=
   //  "DB_PARAMETERS_TEACH"."TEACH SCREEN VALUES";
     "DB_PARAMETERS_TEACH".HMI_PAGE_CONTROL.SAVE_CHANGES_IN_RECIPE := FALSE;
   END_IF;
END_FUNCTION

ORGANIZATION_BLOCK "02_Warm Restart"   // OB100, LAD, Startup
TITLE = "Complete Restart"
{ S7_Optimized_Access := 'FALSE' }
AUTHOR : RCS
// 1.该部分用户可以根据系统的需要将CPU第一次扫描需要执行的逻辑写在此处
// stored: AutoNumber false, SetENOAutomatically false
   VAR_TEMP
      OB100_EV_CLASS : Byte;   // 16#13, Event class 1, Entering event state, Event logged in diagnostic buffer
      OB100_STRTUP : Byte;   // 16#81/82/83/84 Method of startup
      OB100_PRIORITY : Byte;   // Priority of OB Execution
      OB100_OB_NUMBR : Byte;   // 100 (Organization block 100, OB100)
      OB100_RESERVED_1 : Byte;   // Reserved for system
      OB100_RESERVED_2 : Byte;   // Reserved for system
      OB100_STOP : Word;   // Event that caused CPU to stop (16#4xxx)
      OB100_STRT_INFO : DWord;   // Information on how system started
      OB100_DATE_TIME : Date_And_Time;   // Date and time OB100 started
   END_VAR
BEGIN

REGION Network 1
   // 系统程序段无需改动
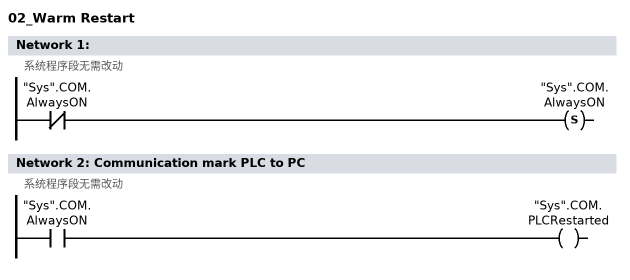
   RUNG wire#powerrail
      I_Contact( "Sys".COM.AlwaysON )
      S_Coil( "Sys".COM.AlwaysON )
   END_RUNG
   // the same network as SCL:
   IF NOT "Sys".COM.AlwaysON THEN "Sys".COM.AlwaysON := TRUE; END_IF;
END_REGION

REGION Network 2: Communication mark PLC to PC
   // 系统程序段无需改动
   RUNG wire#powerrail
      Contact( "Sys".COM.AlwaysON )
      Coil( "Sys".COM.PLCRestarted )
   END_RUNG
   // the same network as SCL:
   "Sys".COM.PLCRestarted := "Sys".COM.AlwaysON;
END_REGION

NETWORK
TITLE = 

      L     1;
      T     "Station_Sys".Status.ModeSV;

END_ORGANIZATION_BLOCK

ORGANIZATION_BLOCK "03_CYC_INT2"   // OB32, LAD, CyclicInterrupt
TITLE = "Cyclic Interrupt"
{ S7_Optimized_Access := 'FALSE' }
VERSION : 0.1
// stored: AutoNumber false, IsIECCheckEnabled false, SetENOAutomatically false
   VAR_TEMP
      OB32_EV_CLASS : Byte;   // Bits 0-3 = 1 (Coming event), Bits 4-7 = 1 (Event class 1)
      OB32_STRT_INF : Byte;   // 16#33 (OB 32 has started)
      OB32_PRIORITY : Byte;   // Priority of OB Execution
      OB32_OB_NUMBR : Byte;   // 32 (Organization block 32, OB32)
      OB32_RESERVED_1 : Byte;   // Reserved for system
      OB32_RESERVED_2 : Byte;   // Reserved for system
      OB32_PHS_OFFSET : Int;   // Phase offset (integer, milliseconds)
      OB32_RESERVED_3 : Int;   // Reserved for system
      OB32_EXC_FREQ : Int;   // Frequency of execution (msec)
      OB32_DATE_TIME : Date_And_Time;   // Date and time OB32 started
   END_VAR
BEGIN

REGION Network 1
   // //Keep resource code
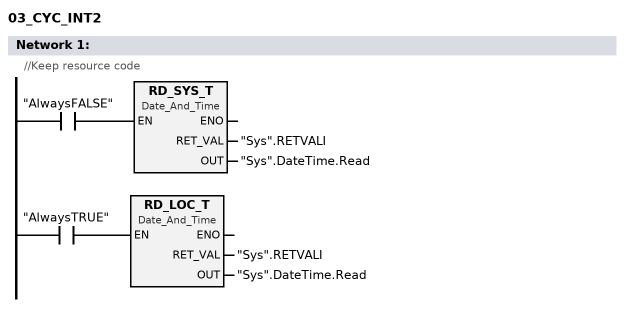
   RUNG wire#powerrail
      Contact( "AlwaysFALSE" )
      { S7_Templates := "date_type := Date_And_Time" } RD_SYS_T(RET_VAL => "Sys".RETVALI, OUT => "Sys".DateTime.Read)
   END_RUNG
   RUNG wire#powerrail
      Contact( "AlwaysTRUE" )
      { S7_Templates := "date_type := Date_And_Time" } RD_LOC_T(RET_VAL => "Sys".RETVALI, OUT => "Sys".DateTime.Read)
   END_RUNG
   // the same network as SCL:
   IF "AlwaysFALSE" THEN "Sys".RETVALI := RD_SYS_T(OUT => "Sys".DateTime.Read); END_IF;
   IF "AlwaysTRUE" THEN "Sys".RETVALI := RD_LOC_T(OUT => "Sys".DateTime.Read); END_IF;
END_REGION

NETWORK
TITLE = Diagnostic
//      CALL  "Diagnostic"
//         iCPUType :=2
//         iDBNum   :=3001
//         iOffset  :=0


END_ORGANIZATION_BLOCK

ORGANIZATION_BLOCK "04_CYC_INT5"   // OB35, LAD, CyclicInterrupt
TITLE = "Cyclic Interrupt"
{ S7_Optimized_Access := 'FALSE' }
VERSION : 0.1
// stored: AutoNumber false, IsIECCheckEnabled false, SetENOAutomatically false
   VAR_TEMP
      OB35_EV_CLASS : Byte;   // Bits 0-3 = 1 (Coming event), Bits 4-7 = 1 (Event class 1)
      OB35_STRT_INF : Byte;   // 16#36 (OB 35 has started)
      OB35_PRIORITY : Byte;   // Priority of OB Execution
      OB35_OB_NUMBR : Byte;   // 35 (Organization block 35, OB35)
      OB35_RESERVED_1 : Byte;   // Reserved for system
      OB35_RESERVED_2 : Byte;   // Reserved for system
      OB35_PHASE_OFFSET : Word;   // Phase offset (msec)
      OB35_RESERVED_3 : Int;   // Reserved for system
      OB35_EXC_FREQ : Int;   // Frequency of execution (msec)
      OB35_DATE_TIME : Date_And_Time;   // Date and time OB35 started
   END_VAR
BEGIN
END_ORGANIZATION_BLOCK

ORGANIZATION_BLOCK "05_MOD_ERR"   // OB122, STL, IOAccessError
TITLE = "Module Access Error"
{ S7_Optimized_Access := 'FALSE' }
   VAR_TEMP
      OB122_EV_CLASS : Byte;   // 16#29, Event class 2, Entering event state, Internal fault event
      OB122_SW_FLT : Byte;   // 16#XX Software error code
      OB122_PRIORITY : Byte;   // Priority of OB Execution
      OB122_OB_NUMBR : Byte;   // 122 (Organization block 122, OB122)
      OB122_BLK_TYPE : Byte;   // 16#88/8C/8E Type of block fault occured in
      OB122_MEM_AREA : Byte;   // Memory area where access error occured
      OB122_MEM_ADDR : Word;   // Memory address where access error occured
      OB122_BLK_NUM : Word;   // Block number in which error occured
      OB122_PRG_ADDR : Word;   // Program address where error occured
      OB122_DATE_TIME : Date_And_Time;   // Date and time OB1 started
   END_VAR
BEGIN
END_ORGANIZATION_BLOCK

ORGANIZATION_BLOCK "07_CYCL_FLT"   // OB80, STL, TimeErrorInterrupt
TITLE = "Cycle Time Fault"
{ S7_Optimized_Access := 'FALSE' }
   VAR_TEMP
      OB80_EV_CLASS : Byte;   // 16#35, Event class 3, Entering event state, Internal fault event
      OB80_FLT_ID : Byte;   // 16#XX, Fault identifcation code
      OB80_PRIORITY : Byte;   // Priority of OB Execution
      OB80_OB_NUMBR : Byte;   // 80 (Organization block 80, OB80)
      OB80_RESERVED_1 : Byte;   // Reserved for system
      OB80_RESERVED_2 : Byte;   // Reserved for system
      OB80_ERROR_INFO : Word;   // Error information on event
      OB80_ERR_EV_CLASS : Byte;   // Class of event causing error
      OB80_ERR_EV_NUM : Byte;   // Number of event causing error
      OB80_OB_PRIORITY : Byte;   // Priority of OB causing error
      OB80_OB_NUM : Byte;   // Number of OB causing error
      OB80_DATE_TIME : Date_And_Time;   // Date and time OB80 started
   END_VAR
BEGIN
END_ORGANIZATION_BLOCK

ORGANIZATION_BLOCK "08_HW_INT0"   // OB40, LAD, HardwareInterrupt
TITLE = "Hardware Interrupt"
{ S7_Optimized_Access := 'FALSE' }
// stored: AutoNumber false, SetENOAutomatically false
   VAR_TEMP
      OB40_EV_CLASS : Byte;   // Bits 0-3 = 1 (Coming event), Bits 4-7 = 1 (Event class 1)
      OB40_STRT_INF : Byte;   // 16#41 (OB 40 has started)
      OB40_PRIORITY : Byte;   // Priority of OB Execution
      OB40_OB_NUMBR : Byte;   // 40 (Organization block 40, OB40)
      OB40_RESERVED_1 : Byte;   // Reserved for system
      OB40_IO_FLAG : Byte;   // 16#54 (input module), 16#55 (output module)
      OB40_MDL_ADDR : Word;   // Base address of module initiating interrupt
      OB40_POINT_ADDR : DWord;   // Interrupt status of the module
      OB40_DATE_TIME : Date_And_Time;   // Date and time OB40 started
   END_VAR
BEGIN
END_ORGANIZATION_BLOCK

ORGANIZATION_BLOCK "09_I/O_FLT1"   // OB82, STL, DiagnosticErrorInterrupt
TITLE = "I/O Point Fault"
{ S7_Optimized_Access := 'FALSE' }
   VAR_TEMP
      OB82_EV_CLASS : Byte;   // 16#39, Event class 3, Entering event state, Internal fault event
      OB82_FLT_ID : Byte;   // 16#XX, Fault identifcation code
      OB82_PRIORITY : Byte;   // Priority of OB Execution
      OB82_OB_NUMBR : Byte;   // 82 (Organization block 82, OB82)
      OB82_RESERVED_1 : Byte;   // Reserved for system
      OB82_IO_FLAG : Byte;   // Input (01010100), Output (01010101)
      OB82_MDL_ADDR : Int;   // Base address of module with fault
      OB82_MDL_DEFECT : Bool;   // Module defective
      OB82_INT_FAULT : Bool;   // Internal fault
      OB82_EXT_FAULT : Bool;   // External fault
      OB82_PNT_INFO : Bool;   // Point information
      OB82_EXT_VOLTAGE : Bool;   // External voltage low
      OB82_FLD_CONNCTR : Bool;   // Field wiring connector missing
      OB82_NO_CONFIG : Bool;   // Module has no configuration data
      OB82_CONFIG_ERR : Bool;   // Module has configuration error
      OB82_MDL_TYPE : Byte;   // Type of module
      OB82_SUB_NDL_ERR : Bool;   // Sub-Module is missing or has error
      OB82_COMM_FAULT : Bool;   // Communication fault
      OB82_MDL_STOP : Bool;   // Module is stopped
      OB82_WTCH_DOG_FLT : Bool;   // Watch dog timer stopped module
      OB82_INT_PS_FLT : Bool;   // Internal power supply fault
      OB82_PRIM_BATT_FLT : Bool;   // Primary battery is in fault
      OB82_BCKUP_BATT_FLT : Bool;   // Backup battery is in fault
      OB82_RESERVED_2 : Bool;   // Reserved for system
      OB82_RACK_FLT : Bool;   // Rack fault, only for bus interface module
      OB82_PROC_FLT : Bool;   // Processor fault
      OB82_EPROM_FLT : Bool;   // EPROM fault
      OB82_RAM_FLT : Bool;   // RAM fault
      OB82_ADU_FLT : Bool;   // ADU fault
      OB82_FUSE_FLT : Bool;   // Fuse fault
      OB82_HW_INTR_FLT : Bool;   // Hardware interupt input in fault
      OB82_RESERVED_3 : Bool;   // Reserved for system
      OB82_DATE_TIME : Date_And_Time;   // Date and time OB82 started
   END_VAR
BEGIN
END_ORGANIZATION_BLOCK

